// TIA Portal V15.1 export
// export: Created 2020-12-23T12:53:55.1483535Z, ExportSetting WithDefaults, WithReadOnly, DisplayName Totally Integrated Automation Portal, DisplayVersion V15.1 Update 3, DisplayName TIA Portal Openness, DisplayVersion V15.1, DisplayName STEP 7 Professional, DisplayVersion V15.1 Update 3, DisplayName WinCC Advanced, DisplayVersion V15.1 Update 3
FUNCTION "func_outputs" : Void   // FC1331, LAD
TITLE = OUTPUTS
{ S7_Optimized_Access := 'TRUE' }
VERSION : 0.1
// stored: AutoNumber false, CodeModifiedDate 2020-12-23T12:53:21.0067533Z, CompileDate 2020-12-23T12:53:51.673862Z, CreationDate 2020-12-23T07:31:02.6354064Z, HandleErrorsWithinBlock false, InterfaceModifiedDate 2020-12-23T12:48:47.2749857Z, IsConsistent true, IsIECCheckEnabled false, IsKnowHowProtected false, IsWriteProtected false, LibraryConformanceStatus The object is library-conformant., ModifiedDate 2020-12-23T12:53:38.1882563Z, ParameterModified 2020-12-23T07:31:02.6354064Z, PLCSimAdvancedSupport false, SetENOAutomatically False, StructureModified 2020-12-23T07:31:02.6354064Z, UDAEnableTagReadback false
BEGIN

REGION Network 1: ------ [1] TBL TABLE LH ------
   // TABLE LH
END_REGION

REGION Network 2: TBL TABLE LH HP UP
   // CONDICIONES DE SEGURIDAD / WARUNKI BEZPIECZENSTWA
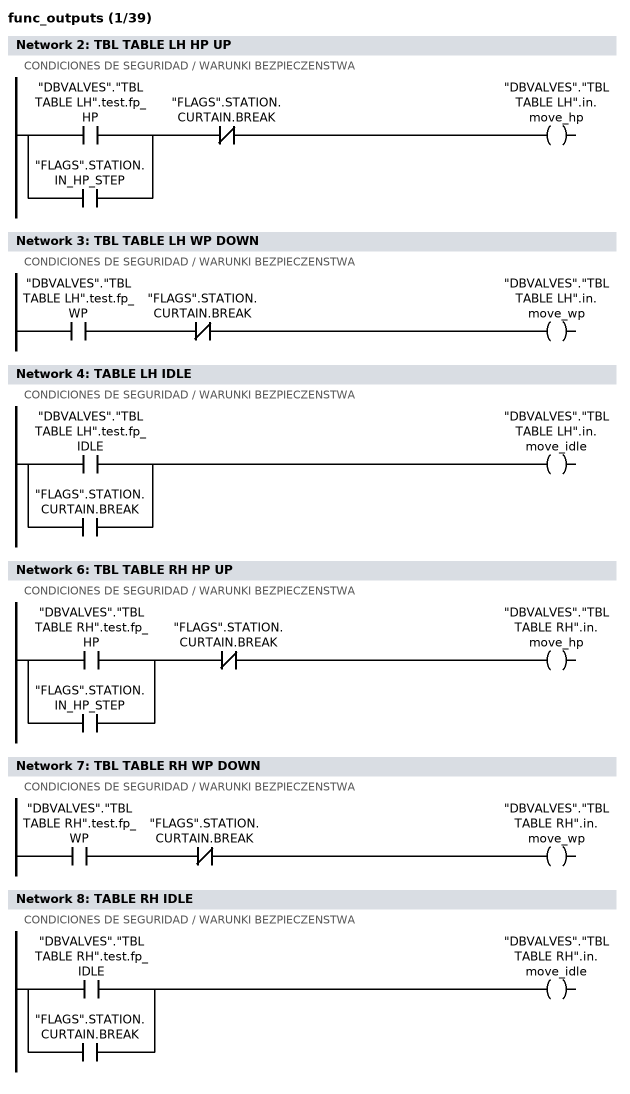
   RUNG wire#powerrail
      Contact( "DBVALVES"."TBL TABLE LH".test.fp_HP )
      wire#w1
      I_Contact( "FLAGS".STATION.CURTAIN.BREAK )
      Coil( "DBVALVES"."TBL TABLE LH".in.move_hp )
   END_RUNG
   RUNG wire#powerrail
      Contact( "FLAGS".STATION.IN_HP_STEP )
   END_RUNG wire#w1
   // the same network as SCL:
   "DBVALVES"."TBL TABLE LH".in.move_hp := ("DBVALVES"."TBL TABLE LH".test.fp_HP OR "FLAGS".STATION.IN_HP_STEP) AND NOT "FLAGS".STATION.CURTAIN.BREAK;
END_REGION

REGION Network 3: TBL TABLE LH WP DOWN
   // CONDICIONES DE SEGURIDAD / WARUNKI BEZPIECZENSTWA
   RUNG wire#powerrail
      Contact( "DBVALVES"."TBL TABLE LH".test.fp_WP )
      I_Contact( "FLAGS".STATION.CURTAIN.BREAK )
      Coil( "DBVALVES"."TBL TABLE LH".in.move_wp )
   END_RUNG
   // the same network as SCL:
   "DBVALVES"."TBL TABLE LH".in.move_wp := "DBVALVES"."TBL TABLE LH".test.fp_WP AND NOT "FLAGS".STATION.CURTAIN.BREAK;
END_REGION

REGION Network 4: TABLE LH IDLE
   // CONDICIONES DE SEGURIDAD / WARUNKI BEZPIECZENSTWA
   RUNG wire#powerrail
      Contact( "DBVALVES"."TBL TABLE LH".test.fp_IDLE )
      wire#w1
      Coil( "DBVALVES"."TBL TABLE LH".in.move_idle )
   END_RUNG
   RUNG wire#powerrail
      Contact( "FLAGS".STATION.CURTAIN.BREAK )
   END_RUNG wire#w1
   // the same network as SCL:
   "DBVALVES"."TBL TABLE LH".in.move_idle := "DBVALVES"."TBL TABLE LH".test.fp_IDLE OR "FLAGS".STATION.CURTAIN.BREAK;
END_REGION

REGION Network 5: ------ [2] TBL TABLE RH ------
   // TABLE RH
END_REGION

REGION Network 6: TBL TABLE RH HP UP
   // CONDICIONES DE SEGURIDAD / WARUNKI BEZPIECZENSTWA
   RUNG wire#powerrail
      Contact( "DBVALVES"."TBL TABLE RH".test.fp_HP )
      wire#w1
      I_Contact( "FLAGS".STATION.CURTAIN.BREAK )
      Coil( "DBVALVES"."TBL TABLE RH".in.move_hp )
   END_RUNG
   RUNG wire#powerrail
      Contact( "FLAGS".STATION.IN_HP_STEP )
   END_RUNG wire#w1
   // the same network as SCL:
   "DBVALVES"."TBL TABLE RH".in.move_hp := ("DBVALVES"."TBL TABLE RH".test.fp_HP OR "FLAGS".STATION.IN_HP_STEP) AND NOT "FLAGS".STATION.CURTAIN.BREAK;
END_REGION

REGION Network 7: TBL TABLE RH WP DOWN
   // CONDICIONES DE SEGURIDAD / WARUNKI BEZPIECZENSTWA
   RUNG wire#powerrail
      Contact( "DBVALVES"."TBL TABLE RH".test.fp_WP )
      I_Contact( "FLAGS".STATION.CURTAIN.BREAK )
      Coil( "DBVALVES"."TBL TABLE RH".in.move_wp )
   END_RUNG
   // the same network as SCL:
   "DBVALVES"."TBL TABLE RH".in.move_wp := "DBVALVES"."TBL TABLE RH".test.fp_WP AND NOT "FLAGS".STATION.CURTAIN.BREAK;
END_REGION

REGION Network 8: TABLE RH IDLE
   // CONDICIONES DE SEGURIDAD / WARUNKI BEZPIECZENSTWA
   RUNG wire#powerrail
      Contact( "DBVALVES"."TBL TABLE RH".test.fp_IDLE )
      wire#w1
      Coil( "DBVALVES"."TBL TABLE RH".in.move_idle )
   END_RUNG
   RUNG wire#powerrail
      Contact( "FLAGS".STATION.CURTAIN.BREAK )
   END_RUNG wire#w1
   // the same network as SCL:
   "DBVALVES"."TBL TABLE RH".in.move_idle := "DBVALVES"."TBL TABLE RH".test.fp_IDLE OR "FLAGS".STATION.CURTAIN.BREAK;
END_REGION

REGION Network 9: ------ [3] TBL SECTION1 ------
   // SECTION1
END_REGION

REGION Network 10: TBL SECTION1 HP UP
   // CONDICIONES DE SEGURIDAD / WARUNKI BEZPIECZENSTWA
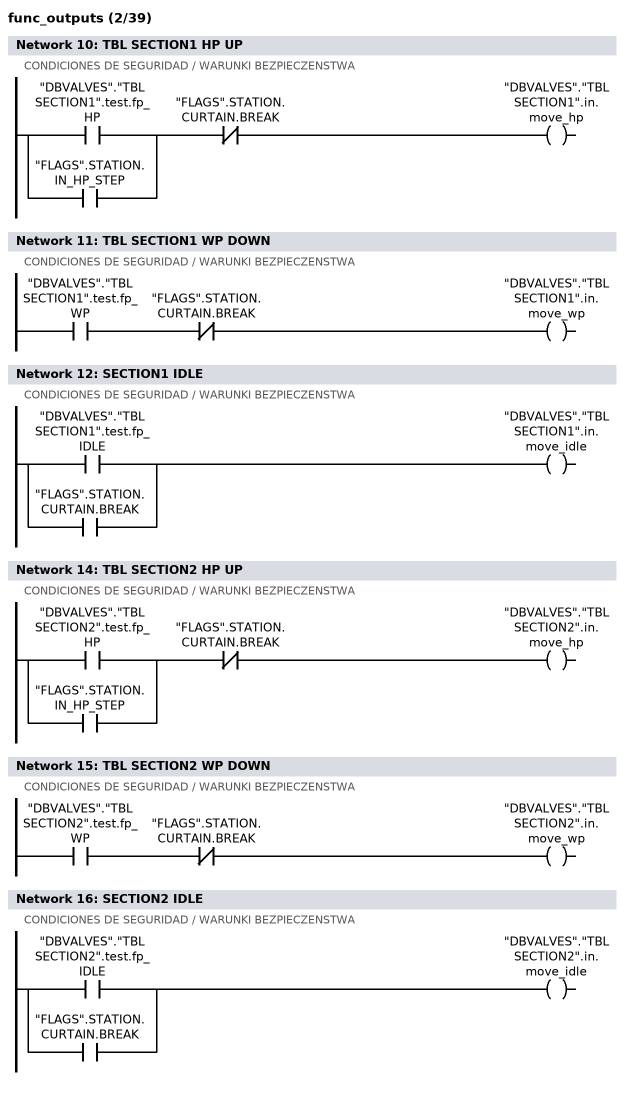
   RUNG wire#powerrail
      Contact( "DBVALVES"."TBL SECTION1".test.fp_HP )
      wire#w1
      I_Contact( "FLAGS".STATION.CURTAIN.BREAK )
      Coil( "DBVALVES"."TBL SECTION1".in.move_hp )
   END_RUNG
   RUNG wire#powerrail
      Contact( "FLAGS".STATION.IN_HP_STEP )
   END_RUNG wire#w1
   // the same network as SCL:
   "DBVALVES"."TBL SECTION1".in.move_hp := ("DBVALVES"."TBL SECTION1".test.fp_HP OR "FLAGS".STATION.IN_HP_STEP) AND NOT "FLAGS".STATION.CURTAIN.BREAK;
END_REGION

REGION Network 11: TBL SECTION1 WP DOWN
   // CONDICIONES DE SEGURIDAD / WARUNKI BEZPIECZENSTWA
   RUNG wire#powerrail
      Contact( "DBVALVES"."TBL SECTION1".test.fp_WP )
      I_Contact( "FLAGS".STATION.CURTAIN.BREAK )
      Coil( "DBVALVES"."TBL SECTION1".in.move_wp )
   END_RUNG
   // the same network as SCL:
   "DBVALVES"."TBL SECTION1".in.move_wp := "DBVALVES"."TBL SECTION1".test.fp_WP AND NOT "FLAGS".STATION.CURTAIN.BREAK;
END_REGION

REGION Network 12: SECTION1 IDLE
   // CONDICIONES DE SEGURIDAD / WARUNKI BEZPIECZENSTWA
   RUNG wire#powerrail
      Contact( "DBVALVES"."TBL SECTION1".test.fp_IDLE )
      wire#w1
      Coil( "DBVALVES"."TBL SECTION1".in.move_idle )
   END_RUNG
   RUNG wire#powerrail
      Contact( "FLAGS".STATION.CURTAIN.BREAK )
   END_RUNG wire#w1
   // the same network as SCL:
   "DBVALVES"."TBL SECTION1".in.move_idle := "DBVALVES"."TBL SECTION1".test.fp_IDLE OR "FLAGS".STATION.CURTAIN.BREAK;
END_REGION

REGION Network 13: ------ [4] TBL SECTION2 ------
   // SECTION2
END_REGION

REGION Network 14: TBL SECTION2 HP UP
   // CONDICIONES DE SEGURIDAD / WARUNKI BEZPIECZENSTWA
   RUNG wire#powerrail
      Contact( "DBVALVES"."TBL SECTION2".test.fp_HP )
      wire#w1
      I_Contact( "FLAGS".STATION.CURTAIN.BREAK )
      Coil( "DBVALVES"."TBL SECTION2".in.move_hp )
   END_RUNG
   RUNG wire#powerrail
      Contact( "FLAGS".STATION.IN_HP_STEP )
   END_RUNG wire#w1
   // the same network as SCL:
   "DBVALVES"."TBL SECTION2".in.move_hp := ("DBVALVES"."TBL SECTION2".test.fp_HP OR "FLAGS".STATION.IN_HP_STEP) AND NOT "FLAGS".STATION.CURTAIN.BREAK;
END_REGION

REGION Network 15: TBL SECTION2 WP DOWN
   // CONDICIONES DE SEGURIDAD / WARUNKI BEZPIECZENSTWA
   RUNG wire#powerrail
      Contact( "DBVALVES"."TBL SECTION2".test.fp_WP )
      I_Contact( "FLAGS".STATION.CURTAIN.BREAK )
      Coil( "DBVALVES"."TBL SECTION2".in.move_wp )
   END_RUNG
   // the same network as SCL:
   "DBVALVES"."TBL SECTION2".in.move_wp := "DBVALVES"."TBL SECTION2".test.fp_WP AND NOT "FLAGS".STATION.CURTAIN.BREAK;
END_REGION

REGION Network 16: SECTION2 IDLE
   // CONDICIONES DE SEGURIDAD / WARUNKI BEZPIECZENSTWA
   RUNG wire#powerrail
      Contact( "DBVALVES"."TBL SECTION2".test.fp_IDLE )
      wire#w1
      Coil( "DBVALVES"."TBL SECTION2".in.move_idle )
   END_RUNG
   RUNG wire#powerrail
      Contact( "FLAGS".STATION.CURTAIN.BREAK )
   END_RUNG wire#w1
   // the same network as SCL:
   "DBVALVES"."TBL SECTION2".in.move_idle := "DBVALVES"."TBL SECTION2".test.fp_IDLE OR "FLAGS".STATION.CURTAIN.BREAK;
END_REGION

REGION Network 17: ------ [5] TBL SECTION4 LH ------
   // SECTION4 LH
END_REGION

REGION Network 18: TBL SECTION4 LH HP UP
   // CONDICIONES DE SEGURIDAD / WARUNKI BEZPIECZENSTWA
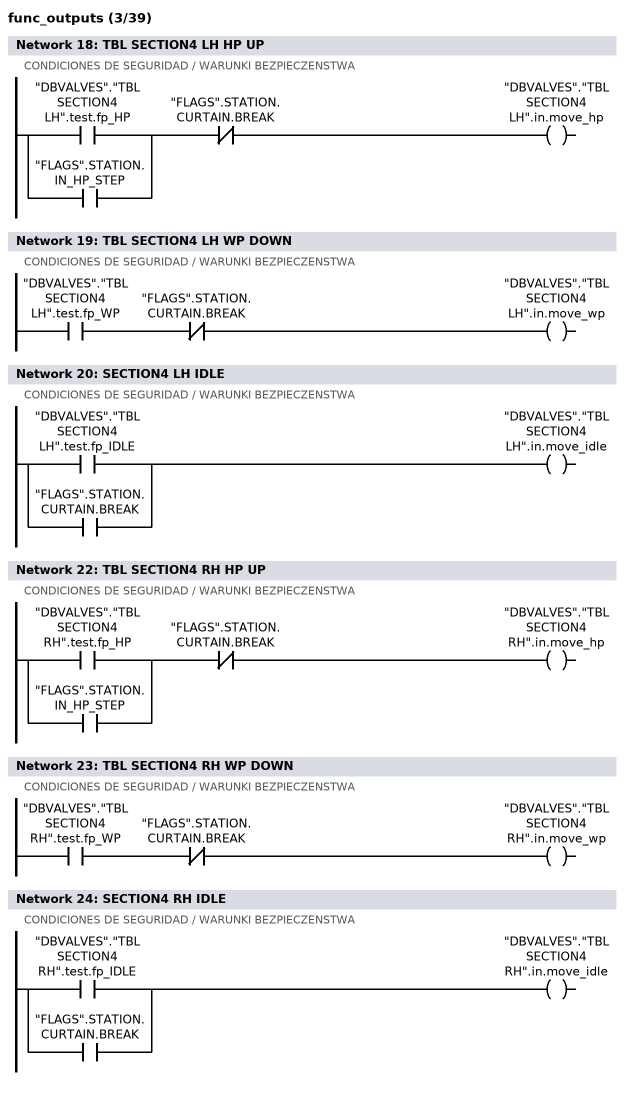
   RUNG wire#powerrail
      Contact( "DBVALVES"."TBL SECTION4 LH".test.fp_HP )
      wire#w1
      I_Contact( "FLAGS".STATION.CURTAIN.BREAK )
      Coil( "DBVALVES"."TBL SECTION4 LH".in.move_hp )
   END_RUNG
   RUNG wire#powerrail
      Contact( "FLAGS".STATION.IN_HP_STEP )
   END_RUNG wire#w1
   // the same network as SCL:
   "DBVALVES"."TBL SECTION4 LH".in.move_hp := ("DBVALVES"."TBL SECTION4 LH".test.fp_HP OR "FLAGS".STATION.IN_HP_STEP) AND NOT "FLAGS".STATION.CURTAIN.BREAK;
END_REGION

REGION Network 19: TBL SECTION4 LH WP DOWN
   // CONDICIONES DE SEGURIDAD / WARUNKI BEZPIECZENSTWA
   RUNG wire#powerrail
      Contact( "DBVALVES"."TBL SECTION4 LH".test.fp_WP )
      I_Contact( "FLAGS".STATION.CURTAIN.BREAK )
      Coil( "DBVALVES"."TBL SECTION4 LH".in.move_wp )
   END_RUNG
   // the same network as SCL:
   "DBVALVES"."TBL SECTION4 LH".in.move_wp := "DBVALVES"."TBL SECTION4 LH".test.fp_WP AND NOT "FLAGS".STATION.CURTAIN.BREAK;
END_REGION

REGION Network 20: SECTION4 LH IDLE
   // CONDICIONES DE SEGURIDAD / WARUNKI BEZPIECZENSTWA
   RUNG wire#powerrail
      Contact( "DBVALVES"."TBL SECTION4 LH".test.fp_IDLE )
      wire#w1
      Coil( "DBVALVES"."TBL SECTION4 LH".in.move_idle )
   END_RUNG
   RUNG wire#powerrail
      Contact( "FLAGS".STATION.CURTAIN.BREAK )
   END_RUNG wire#w1
   // the same network as SCL:
   "DBVALVES"."TBL SECTION4 LH".in.move_idle := "DBVALVES"."TBL SECTION4 LH".test.fp_IDLE OR "FLAGS".STATION.CURTAIN.BREAK;
END_REGION

REGION Network 21: ------ [6] TBL SECTION4 RH ------
   // SECTION4 RH
END_REGION

REGION Network 22: TBL SECTION4 RH HP UP
   // CONDICIONES DE SEGURIDAD / WARUNKI BEZPIECZENSTWA
   RUNG wire#powerrail
      Contact( "DBVALVES"."TBL SECTION4 RH".test.fp_HP )
      wire#w1
      I_Contact( "FLAGS".STATION.CURTAIN.BREAK )
      Coil( "DBVALVES"."TBL SECTION4 RH".in.move_hp )
   END_RUNG
   RUNG wire#powerrail
      Contact( "FLAGS".STATION.IN_HP_STEP )
   END_RUNG wire#w1
   // the same network as SCL:
   "DBVALVES"."TBL SECTION4 RH".in.move_hp := ("DBVALVES"."TBL SECTION4 RH".test.fp_HP OR "FLAGS".STATION.IN_HP_STEP) AND NOT "FLAGS".STATION.CURTAIN.BREAK;
END_REGION

REGION Network 23: TBL SECTION4 RH WP DOWN
   // CONDICIONES DE SEGURIDAD / WARUNKI BEZPIECZENSTWA
   RUNG wire#powerrail
      Contact( "DBVALVES"."TBL SECTION4 RH".test.fp_WP )
      I_Contact( "FLAGS".STATION.CURTAIN.BREAK )
      Coil( "DBVALVES"."TBL SECTION4 RH".in.move_wp )
   END_RUNG
   // the same network as SCL:
   "DBVALVES"."TBL SECTION4 RH".in.move_wp := "DBVALVES"."TBL SECTION4 RH".test.fp_WP AND NOT "FLAGS".STATION.CURTAIN.BREAK;
END_REGION

REGION Network 24: SECTION4 RH IDLE
   // CONDICIONES DE SEGURIDAD / WARUNKI BEZPIECZENSTWA
   RUNG wire#powerrail
      Contact( "DBVALVES"."TBL SECTION4 RH".test.fp_IDLE )
      wire#w1
      Coil( "DBVALVES"."TBL SECTION4 RH".in.move_idle )
   END_RUNG
   RUNG wire#powerrail
      Contact( "FLAGS".STATION.CURTAIN.BREAK )
   END_RUNG wire#w1
   // the same network as SCL:
   "DBVALVES"."TBL SECTION4 RH".in.move_idle := "DBVALVES"."TBL SECTION4 RH".test.fp_IDLE OR "FLAGS".STATION.CURTAIN.BREAK;
END_REGION

REGION Network 25: ------ [7] TBL SECTION5 LH ------
   // SECTION5 LH
END_REGION

REGION Network 26: TBL SECTION5 LH HP UP
   // CONDICIONES DE SEGURIDAD / WARUNKI BEZPIECZENSTWA
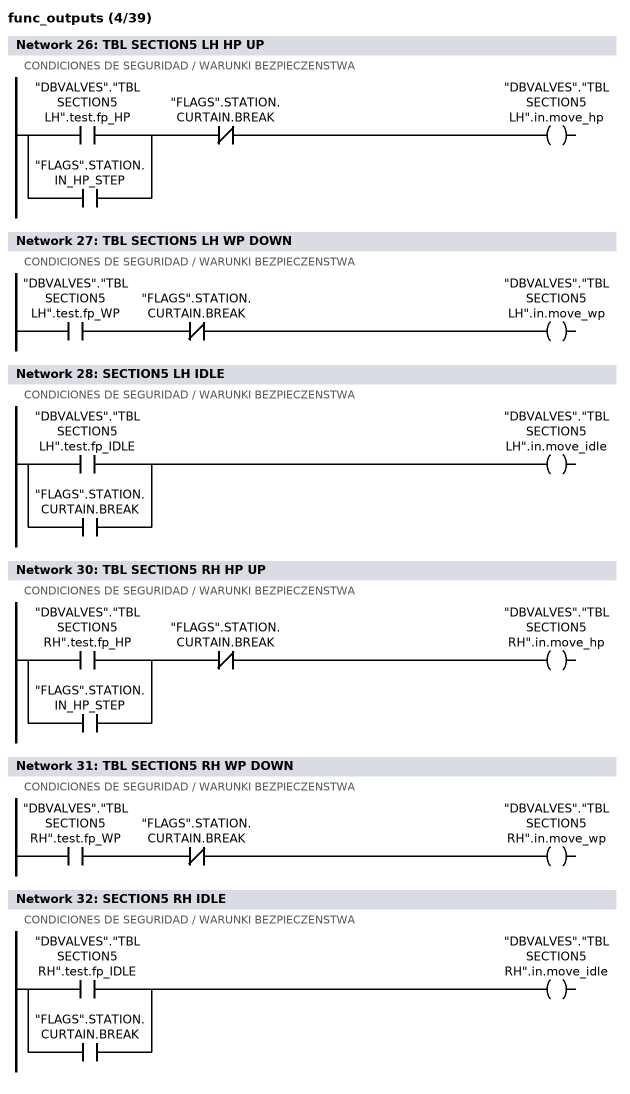
   RUNG wire#powerrail
      Contact( "DBVALVES"."TBL SECTION5 LH".test.fp_HP )
      wire#w1
      I_Contact( "FLAGS".STATION.CURTAIN.BREAK )
      Coil( "DBVALVES"."TBL SECTION5 LH".in.move_hp )
   END_RUNG
   RUNG wire#powerrail
      Contact( "FLAGS".STATION.IN_HP_STEP )
   END_RUNG wire#w1
   // the same network as SCL:
   "DBVALVES"."TBL SECTION5 LH".in.move_hp := ("DBVALVES"."TBL SECTION5 LH".test.fp_HP OR "FLAGS".STATION.IN_HP_STEP) AND NOT "FLAGS".STATION.CURTAIN.BREAK;
END_REGION

REGION Network 27: TBL SECTION5 LH WP DOWN
   // CONDICIONES DE SEGURIDAD / WARUNKI BEZPIECZENSTWA
   RUNG wire#powerrail
      Contact( "DBVALVES"."TBL SECTION5 LH".test.fp_WP )
      I_Contact( "FLAGS".STATION.CURTAIN.BREAK )
      Coil( "DBVALVES"."TBL SECTION5 LH".in.move_wp )
   END_RUNG
   // the same network as SCL:
   "DBVALVES"."TBL SECTION5 LH".in.move_wp := "DBVALVES"."TBL SECTION5 LH".test.fp_WP AND NOT "FLAGS".STATION.CURTAIN.BREAK;
END_REGION

REGION Network 28: SECTION5 LH IDLE
   // CONDICIONES DE SEGURIDAD / WARUNKI BEZPIECZENSTWA
   RUNG wire#powerrail
      Contact( "DBVALVES"."TBL SECTION5 LH".test.fp_IDLE )
      wire#w1
      Coil( "DBVALVES"."TBL SECTION5 LH".in.move_idle )
   END_RUNG
   RUNG wire#powerrail
      Contact( "FLAGS".STATION.CURTAIN.BREAK )
   END_RUNG wire#w1
   // the same network as SCL:
   "DBVALVES"."TBL SECTION5 LH".in.move_idle := "DBVALVES"."TBL SECTION5 LH".test.fp_IDLE OR "FLAGS".STATION.CURTAIN.BREAK;
END_REGION

REGION Network 29: ------ [8] TBL SECTION5 RH ------
   // SECTION5 RH
END_REGION

REGION Network 30: TBL SECTION5 RH HP UP
   // CONDICIONES DE SEGURIDAD / WARUNKI BEZPIECZENSTWA
   RUNG wire#powerrail
      Contact( "DBVALVES"."TBL SECTION5 RH".test.fp_HP )
      wire#w1
      I_Contact( "FLAGS".STATION.CURTAIN.BREAK )
      Coil( "DBVALVES"."TBL SECTION5 RH".in.move_hp )
   END_RUNG
   RUNG wire#powerrail
      Contact( "FLAGS".STATION.IN_HP_STEP )
   END_RUNG wire#w1
   // the same network as SCL:
   "DBVALVES"."TBL SECTION5 RH".in.move_hp := ("DBVALVES"."TBL SECTION5 RH".test.fp_HP OR "FLAGS".STATION.IN_HP_STEP) AND NOT "FLAGS".STATION.CURTAIN.BREAK;
END_REGION

REGION Network 31: TBL SECTION5 RH WP DOWN
   // CONDICIONES DE SEGURIDAD / WARUNKI BEZPIECZENSTWA
   RUNG wire#powerrail
      Contact( "DBVALVES"."TBL SECTION5 RH".test.fp_WP )
      I_Contact( "FLAGS".STATION.CURTAIN.BREAK )
      Coil( "DBVALVES"."TBL SECTION5 RH".in.move_wp )
   END_RUNG
   // the same network as SCL:
   "DBVALVES"."TBL SECTION5 RH".in.move_wp := "DBVALVES"."TBL SECTION5 RH".test.fp_WP AND NOT "FLAGS".STATION.CURTAIN.BREAK;
END_REGION

REGION Network 32: SECTION5 RH IDLE
   // CONDICIONES DE SEGURIDAD / WARUNKI BEZPIECZENSTWA
   RUNG wire#powerrail
      Contact( "DBVALVES"."TBL SECTION5 RH".test.fp_IDLE )
      wire#w1
      Coil( "DBVALVES"."TBL SECTION5 RH".in.move_idle )
   END_RUNG
   RUNG wire#powerrail
      Contact( "FLAGS".STATION.CURTAIN.BREAK )
   END_RUNG wire#w1
   // the same network as SCL:
   "DBVALVES"."TBL SECTION5 RH".in.move_idle := "DBVALVES"."TBL SECTION5 RH".test.fp_IDLE OR "FLAGS".STATION.CURTAIN.BREAK;
END_REGION

REGION Network 33: ------ [9] TBL POSITIONING LH ------
   // POSITIONING LH
END_REGION

REGION Network 34: TBL POSITIONING LH HP UP
   // CONDICIONES DE SEGURIDAD / WARUNKI BEZPIECZENSTWA
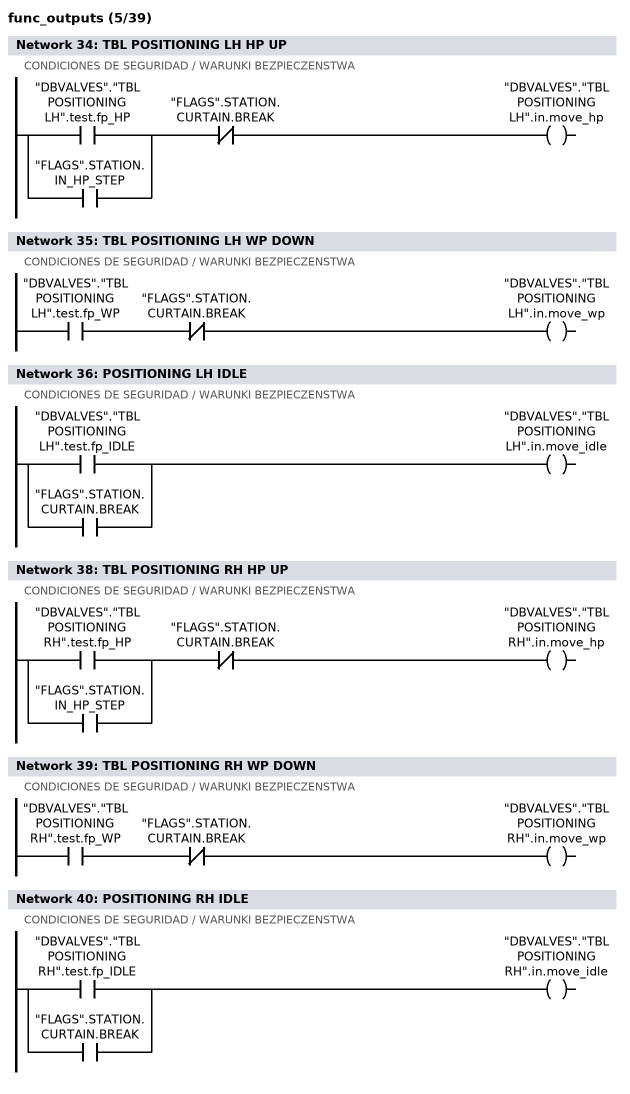
   RUNG wire#powerrail
      Contact( "DBVALVES"."TBL POSITIONING LH".test.fp_HP )
      wire#w1
      I_Contact( "FLAGS".STATION.CURTAIN.BREAK )
      Coil( "DBVALVES"."TBL POSITIONING LH".in.move_hp )
   END_RUNG
   RUNG wire#powerrail
      Contact( "FLAGS".STATION.IN_HP_STEP )
   END_RUNG wire#w1
   // the same network as SCL:
   "DBVALVES"."TBL POSITIONING LH".in.move_hp := ("DBVALVES"."TBL POSITIONING LH".test.fp_HP OR "FLAGS".STATION.IN_HP_STEP) AND NOT "FLAGS".STATION.CURTAIN.BREAK;
END_REGION

REGION Network 35: TBL POSITIONING LH WP DOWN
   // CONDICIONES DE SEGURIDAD / WARUNKI BEZPIECZENSTWA
   RUNG wire#powerrail
      Contact( "DBVALVES"."TBL POSITIONING LH".test.fp_WP )
      I_Contact( "FLAGS".STATION.CURTAIN.BREAK )
      Coil( "DBVALVES"."TBL POSITIONING LH".in.move_wp )
   END_RUNG
   // the same network as SCL:
   "DBVALVES"."TBL POSITIONING LH".in.move_wp := "DBVALVES"."TBL POSITIONING LH".test.fp_WP AND NOT "FLAGS".STATION.CURTAIN.BREAK;
END_REGION

REGION Network 36: POSITIONING LH IDLE
   // CONDICIONES DE SEGURIDAD / WARUNKI BEZPIECZENSTWA
   RUNG wire#powerrail
      Contact( "DBVALVES"."TBL POSITIONING LH".test.fp_IDLE )
      wire#w1
      Coil( "DBVALVES"."TBL POSITIONING LH".in.move_idle )
   END_RUNG
   RUNG wire#powerrail
      Contact( "FLAGS".STATION.CURTAIN.BREAK )
   END_RUNG wire#w1
   // the same network as SCL:
   "DBVALVES"."TBL POSITIONING LH".in.move_idle := "DBVALVES"."TBL POSITIONING LH".test.fp_IDLE OR "FLAGS".STATION.CURTAIN.BREAK;
END_REGION

REGION Network 37: ------ [10] TBL POSITIONING RH ------
   // POSITIONING RH
END_REGION

REGION Network 38: TBL POSITIONING RH HP UP
   // CONDICIONES DE SEGURIDAD / WARUNKI BEZPIECZENSTWA
   RUNG wire#powerrail
      Contact( "DBVALVES"."TBL POSITIONING RH".test.fp_HP )
      wire#w1
      I_Contact( "FLAGS".STATION.CURTAIN.BREAK )
      Coil( "DBVALVES"."TBL POSITIONING RH".in.move_hp )
   END_RUNG
   RUNG wire#powerrail
      Contact( "FLAGS".STATION.IN_HP_STEP )
   END_RUNG wire#w1
   // the same network as SCL:
   "DBVALVES"."TBL POSITIONING RH".in.move_hp := ("DBVALVES"."TBL POSITIONING RH".test.fp_HP OR "FLAGS".STATION.IN_HP_STEP) AND NOT "FLAGS".STATION.CURTAIN.BREAK;
END_REGION

REGION Network 39: TBL POSITIONING RH WP DOWN
   // CONDICIONES DE SEGURIDAD / WARUNKI BEZPIECZENSTWA
   RUNG wire#powerrail
      Contact( "DBVALVES"."TBL POSITIONING RH".test.fp_WP )
      I_Contact( "FLAGS".STATION.CURTAIN.BREAK )
      Coil( "DBVALVES"."TBL POSITIONING RH".in.move_wp )
   END_RUNG
   // the same network as SCL:
   "DBVALVES"."TBL POSITIONING RH".in.move_wp := "DBVALVES"."TBL POSITIONING RH".test.fp_WP AND NOT "FLAGS".STATION.CURTAIN.BREAK;
END_REGION

REGION Network 40: POSITIONING RH IDLE
   // CONDICIONES DE SEGURIDAD / WARUNKI BEZPIECZENSTWA
   RUNG wire#powerrail
      Contact( "DBVALVES"."TBL POSITIONING RH".test.fp_IDLE )
      wire#w1
      Coil( "DBVALVES"."TBL POSITIONING RH".in.move_idle )
   END_RUNG
   RUNG wire#powerrail
      Contact( "FLAGS".STATION.CURTAIN.BREAK )
   END_RUNG wire#w1
   // the same network as SCL:
   "DBVALVES"."TBL POSITIONING RH".in.move_idle := "DBVALVES"."TBL POSITIONING RH".test.fp_IDLE OR "FLAGS".STATION.CURTAIN.BREAK;
END_REGION

REGION Network 41: ------ [11] TBL PIN LH ------
   // PIN LH
END_REGION

REGION Network 42: TBL PIN LH HP DOWN
   // CONDICIONES DE SEGURIDAD / WARUNKI BEZPIECZENSTWA
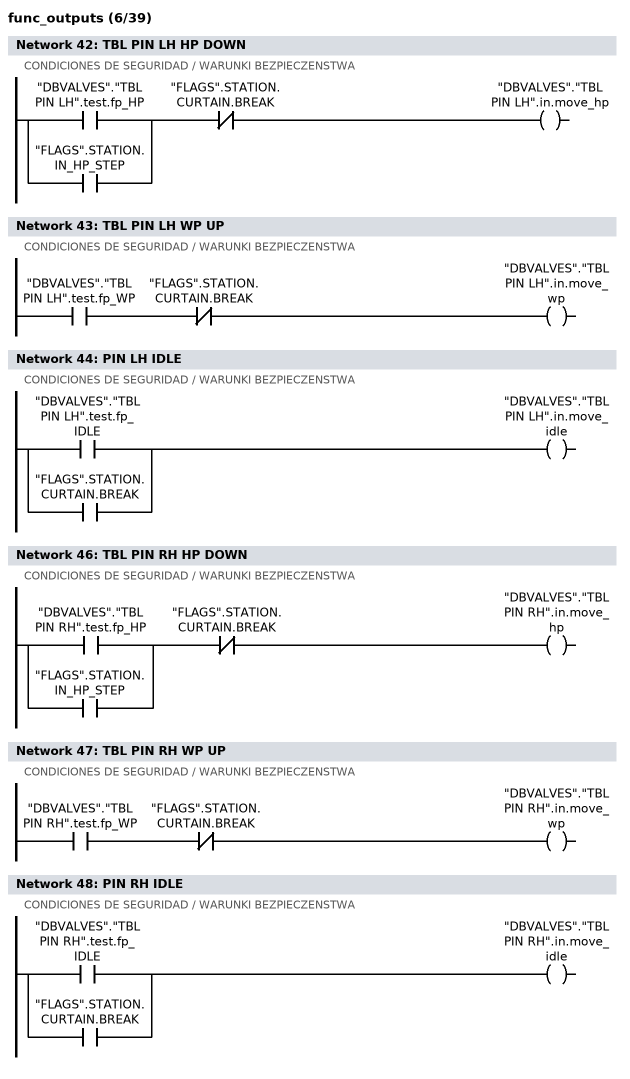
   RUNG wire#powerrail
      Contact( "DBVALVES"."TBL PIN LH".test.fp_HP )
      wire#w1
      I_Contact( "FLAGS".STATION.CURTAIN.BREAK )
      Coil( "DBVALVES"."TBL PIN LH".in.move_hp )
   END_RUNG
   RUNG wire#powerrail
      Contact( "FLAGS".STATION.IN_HP_STEP )
   END_RUNG wire#w1
   // the same network as SCL:
   "DBVALVES"."TBL PIN LH".in.move_hp := ("DBVALVES"."TBL PIN LH".test.fp_HP OR "FLAGS".STATION.IN_HP_STEP) AND NOT "FLAGS".STATION.CURTAIN.BREAK;
END_REGION

REGION Network 43: TBL PIN LH WP UP
   // CONDICIONES DE SEGURIDAD / WARUNKI BEZPIECZENSTWA
   RUNG wire#powerrail
      Contact( "DBVALVES"."TBL PIN LH".test.fp_WP )
      I_Contact( "FLAGS".STATION.CURTAIN.BREAK )
      Coil( "DBVALVES"."TBL PIN LH".in.move_wp )
   END_RUNG
   // the same network as SCL:
   "DBVALVES"."TBL PIN LH".in.move_wp := "DBVALVES"."TBL PIN LH".test.fp_WP AND NOT "FLAGS".STATION.CURTAIN.BREAK;
END_REGION

REGION Network 44: PIN LH IDLE
   // CONDICIONES DE SEGURIDAD / WARUNKI BEZPIECZENSTWA
   RUNG wire#powerrail
      Contact( "DBVALVES"."TBL PIN LH".test.fp_IDLE )
      wire#w1
      Coil( "DBVALVES"."TBL PIN LH".in.move_idle )
   END_RUNG
   RUNG wire#powerrail
      Contact( "FLAGS".STATION.CURTAIN.BREAK )
   END_RUNG wire#w1
   // the same network as SCL:
   "DBVALVES"."TBL PIN LH".in.move_idle := "DBVALVES"."TBL PIN LH".test.fp_IDLE OR "FLAGS".STATION.CURTAIN.BREAK;
END_REGION

REGION Network 45: ------ [12] TBL PIN RH ------
   // PIN RH
END_REGION

REGION Network 46: TBL PIN RH HP DOWN
   // CONDICIONES DE SEGURIDAD / WARUNKI BEZPIECZENSTWA
   RUNG wire#powerrail
      Contact( "DBVALVES"."TBL PIN RH".test.fp_HP )
      wire#w1
      I_Contact( "FLAGS".STATION.CURTAIN.BREAK )
      Coil( "DBVALVES"."TBL PIN RH".in.move_hp )
   END_RUNG
   RUNG wire#powerrail
      Contact( "FLAGS".STATION.IN_HP_STEP )
   END_RUNG wire#w1
   // the same network as SCL:
   "DBVALVES"."TBL PIN RH".in.move_hp := ("DBVALVES"."TBL PIN RH".test.fp_HP OR "FLAGS".STATION.IN_HP_STEP) AND NOT "FLAGS".STATION.CURTAIN.BREAK;
END_REGION

REGION Network 47: TBL PIN RH WP UP
   // CONDICIONES DE SEGURIDAD / WARUNKI BEZPIECZENSTWA
   RUNG wire#powerrail
      Contact( "DBVALVES"."TBL PIN RH".test.fp_WP )
      I_Contact( "FLAGS".STATION.CURTAIN.BREAK )
      Coil( "DBVALVES"."TBL PIN RH".in.move_wp )
   END_RUNG
   // the same network as SCL:
   "DBVALVES"."TBL PIN RH".in.move_wp := "DBVALVES"."TBL PIN RH".test.fp_WP AND NOT "FLAGS".STATION.CURTAIN.BREAK;
END_REGION

REGION Network 48: PIN RH IDLE
   // CONDICIONES DE SEGURIDAD / WARUNKI BEZPIECZENSTWA
   RUNG wire#powerrail
      Contact( "DBVALVES"."TBL PIN RH".test.fp_IDLE )
      wire#w1
      Coil( "DBVALVES"."TBL PIN RH".in.move_idle )
   END_RUNG
   RUNG wire#powerrail
      Contact( "FLAGS".STATION.CURTAIN.BREAK )
   END_RUNG wire#w1
   // the same network as SCL:
   "DBVALVES"."TBL PIN RH".in.move_idle := "DBVALVES"."TBL PIN RH".test.fp_IDLE OR "FLAGS".STATION.CURTAIN.BREAK;
END_REGION

REGION Network 49: ------ [13] TBL SCREW GRIPPER ------
   // SCREW GRIPPER
END_REGION

REGION Network 50: TBL SCREW GRIPPER HP OPEN
   // CONDICIONES DE SEGURIDAD / WARUNKI BEZPIECZENSTWA
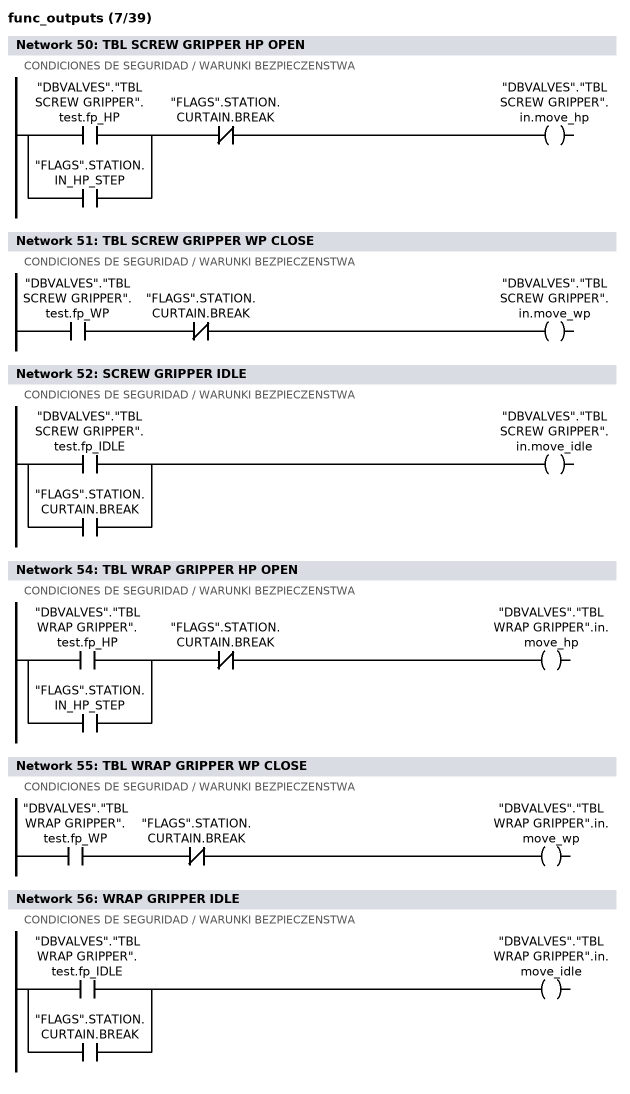
   RUNG wire#powerrail
      Contact( "DBVALVES"."TBL SCREW GRIPPER".test.fp_HP )
      wire#w1
      I_Contact( "FLAGS".STATION.CURTAIN.BREAK )
      Coil( "DBVALVES"."TBL SCREW GRIPPER".in.move_hp )
   END_RUNG
   RUNG wire#powerrail
      Contact( "FLAGS".STATION.IN_HP_STEP )
   END_RUNG wire#w1
   // the same network as SCL:
   "DBVALVES"."TBL SCREW GRIPPER".in.move_hp := ("DBVALVES"."TBL SCREW GRIPPER".test.fp_HP OR "FLAGS".STATION.IN_HP_STEP) AND NOT "FLAGS".STATION.CURTAIN.BREAK;
END_REGION

REGION Network 51: TBL SCREW GRIPPER WP CLOSE
   // CONDICIONES DE SEGURIDAD / WARUNKI BEZPIECZENSTWA
   RUNG wire#powerrail
      Contact( "DBVALVES"."TBL SCREW GRIPPER".test.fp_WP )
      I_Contact( "FLAGS".STATION.CURTAIN.BREAK )
      Coil( "DBVALVES"."TBL SCREW GRIPPER".in.move_wp )
   END_RUNG
   // the same network as SCL:
   "DBVALVES"."TBL SCREW GRIPPER".in.move_wp := "DBVALVES"."TBL SCREW GRIPPER".test.fp_WP AND NOT "FLAGS".STATION.CURTAIN.BREAK;
END_REGION

REGION Network 52: SCREW GRIPPER IDLE
   // CONDICIONES DE SEGURIDAD / WARUNKI BEZPIECZENSTWA
   RUNG wire#powerrail
      Contact( "DBVALVES"."TBL SCREW GRIPPER".test.fp_IDLE )
      wire#w1
      Coil( "DBVALVES"."TBL SCREW GRIPPER".in.move_idle )
   END_RUNG
   RUNG wire#powerrail
      Contact( "FLAGS".STATION.CURTAIN.BREAK )
   END_RUNG wire#w1
   // the same network as SCL:
   "DBVALVES"."TBL SCREW GRIPPER".in.move_idle := "DBVALVES"."TBL SCREW GRIPPER".test.fp_IDLE OR "FLAGS".STATION.CURTAIN.BREAK;
END_REGION

REGION Network 53: ------ [14] TBL WRAP GRIPPER ------
   // WRAP GRIPPER
END_REGION

REGION Network 54: TBL WRAP GRIPPER HP OPEN
   // CONDICIONES DE SEGURIDAD / WARUNKI BEZPIECZENSTWA
   RUNG wire#powerrail
      Contact( "DBVALVES"."TBL WRAP GRIPPER".test.fp_HP )
      wire#w1
      I_Contact( "FLAGS".STATION.CURTAIN.BREAK )
      Coil( "DBVALVES"."TBL WRAP GRIPPER".in.move_hp )
   END_RUNG
   RUNG wire#powerrail
      Contact( "FLAGS".STATION.IN_HP_STEP )
   END_RUNG wire#w1
   // the same network as SCL:
   "DBVALVES"."TBL WRAP GRIPPER".in.move_hp := ("DBVALVES"."TBL WRAP GRIPPER".test.fp_HP OR "FLAGS".STATION.IN_HP_STEP) AND NOT "FLAGS".STATION.CURTAIN.BREAK;
END_REGION

REGION Network 55: TBL WRAP GRIPPER WP CLOSE
   // CONDICIONES DE SEGURIDAD / WARUNKI BEZPIECZENSTWA
   RUNG wire#powerrail
      Contact( "DBVALVES"."TBL WRAP GRIPPER".test.fp_WP )
      I_Contact( "FLAGS".STATION.CURTAIN.BREAK )
      Coil( "DBVALVES"."TBL WRAP GRIPPER".in.move_wp )
   END_RUNG
   // the same network as SCL:
   "DBVALVES"."TBL WRAP GRIPPER".in.move_wp := "DBVALVES"."TBL WRAP GRIPPER".test.fp_WP AND NOT "FLAGS".STATION.CURTAIN.BREAK;
END_REGION

REGION Network 56: WRAP GRIPPER IDLE
   // CONDICIONES DE SEGURIDAD / WARUNKI BEZPIECZENSTWA
   RUNG wire#powerrail
      Contact( "DBVALVES"."TBL WRAP GRIPPER".test.fp_IDLE )
      wire#w1
      Coil( "DBVALVES"."TBL WRAP GRIPPER".in.move_idle )
   END_RUNG
   RUNG wire#powerrail
      Contact( "FLAGS".STATION.CURTAIN.BREAK )
   END_RUNG wire#w1
   // the same network as SCL:
   "DBVALVES"."TBL WRAP GRIPPER".in.move_idle := "DBVALVES"."TBL WRAP GRIPPER".test.fp_IDLE OR "FLAGS".STATION.CURTAIN.BREAK;
END_REGION

REGION Network 57: ------ [15] ST1 POSITIONING ------
   // POSITIONING
END_REGION

REGION Network 58: ST1 POSITIONING HP RIGHT
   // CONDICIONES DE SEGURIDAD / WARUNKI BEZPIECZENSTWA
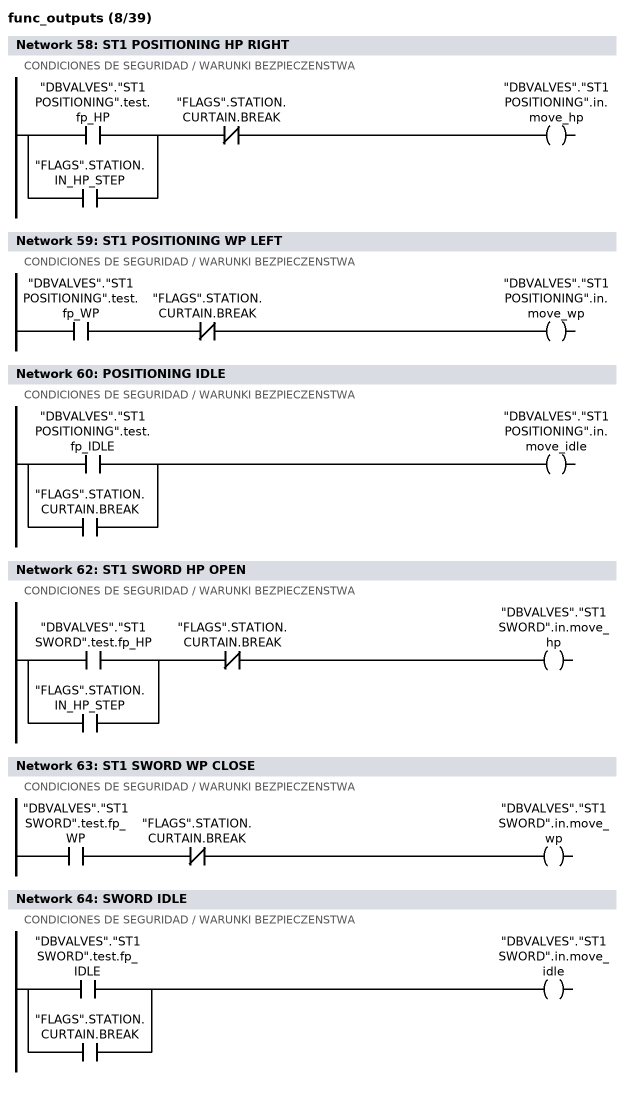
   RUNG wire#powerrail
      Contact( "DBVALVES"."ST1 POSITIONING".test.fp_HP )
      wire#w1
      I_Contact( "FLAGS".STATION.CURTAIN.BREAK )
      Coil( "DBVALVES"."ST1 POSITIONING".in.move_hp )
   END_RUNG
   RUNG wire#powerrail
      Contact( "FLAGS".STATION.IN_HP_STEP )
   END_RUNG wire#w1
   // the same network as SCL:
   "DBVALVES"."ST1 POSITIONING".in.move_hp := ("DBVALVES"."ST1 POSITIONING".test.fp_HP OR "FLAGS".STATION.IN_HP_STEP) AND NOT "FLAGS".STATION.CURTAIN.BREAK;
END_REGION

REGION Network 59: ST1 POSITIONING WP LEFT
   // CONDICIONES DE SEGURIDAD / WARUNKI BEZPIECZENSTWA
   RUNG wire#powerrail
      Contact( "DBVALVES"."ST1 POSITIONING".test.fp_WP )
      I_Contact( "FLAGS".STATION.CURTAIN.BREAK )
      Coil( "DBVALVES"."ST1 POSITIONING".in.move_wp )
   END_RUNG
   // the same network as SCL:
   "DBVALVES"."ST1 POSITIONING".in.move_wp := "DBVALVES"."ST1 POSITIONING".test.fp_WP AND NOT "FLAGS".STATION.CURTAIN.BREAK;
END_REGION

REGION Network 60: POSITIONING IDLE
   // CONDICIONES DE SEGURIDAD / WARUNKI BEZPIECZENSTWA
   RUNG wire#powerrail
      Contact( "DBVALVES"."ST1 POSITIONING".test.fp_IDLE )
      wire#w1
      Coil( "DBVALVES"."ST1 POSITIONING".in.move_idle )
   END_RUNG
   RUNG wire#powerrail
      Contact( "FLAGS".STATION.CURTAIN.BREAK )
   END_RUNG wire#w1
   // the same network as SCL:
   "DBVALVES"."ST1 POSITIONING".in.move_idle := "DBVALVES"."ST1 POSITIONING".test.fp_IDLE OR "FLAGS".STATION.CURTAIN.BREAK;
END_REGION

REGION Network 61: ------ [16] ST1 SWORD ------
   // SWORD
END_REGION

REGION Network 62: ST1 SWORD HP OPEN
   // CONDICIONES DE SEGURIDAD / WARUNKI BEZPIECZENSTWA
   RUNG wire#powerrail
      Contact( "DBVALVES"."ST1 SWORD".test.fp_HP )
      wire#w1
      I_Contact( "FLAGS".STATION.CURTAIN.BREAK )
      Coil( "DBVALVES"."ST1 SWORD".in.move_hp )
   END_RUNG
   RUNG wire#powerrail
      Contact( "FLAGS".STATION.IN_HP_STEP )
   END_RUNG wire#w1
   // the same network as SCL:
   "DBVALVES"."ST1 SWORD".in.move_hp := ("DBVALVES"."ST1 SWORD".test.fp_HP OR "FLAGS".STATION.IN_HP_STEP) AND NOT "FLAGS".STATION.CURTAIN.BREAK;
END_REGION

REGION Network 63: ST1 SWORD WP CLOSE
   // CONDICIONES DE SEGURIDAD / WARUNKI BEZPIECZENSTWA
   RUNG wire#powerrail
      Contact( "DBVALVES"."ST1 SWORD".test.fp_WP )
      I_Contact( "FLAGS".STATION.CURTAIN.BREAK )
      Coil( "DBVALVES"."ST1 SWORD".in.move_wp )
   END_RUNG
   // the same network as SCL:
   "DBVALVES"."ST1 SWORD".in.move_wp := "DBVALVES"."ST1 SWORD".test.fp_WP AND NOT "FLAGS".STATION.CURTAIN.BREAK;
END_REGION

REGION Network 64: SWORD IDLE
   // CONDICIONES DE SEGURIDAD / WARUNKI BEZPIECZENSTWA
   RUNG wire#powerrail
      Contact( "DBVALVES"."ST1 SWORD".test.fp_IDLE )
      wire#w1
      Coil( "DBVALVES"."ST1 SWORD".in.move_idle )
   END_RUNG
   RUNG wire#powerrail
      Contact( "FLAGS".STATION.CURTAIN.BREAK )
   END_RUNG wire#w1
   // the same network as SCL:
   "DBVALVES"."ST1 SWORD".in.move_idle := "DBVALVES"."ST1 SWORD".test.fp_IDLE OR "FLAGS".STATION.CURTAIN.BREAK;
END_REGION

REGION Network 65: ------ [17] ST2 POSITIONING ------
   // POSITIONING
END_REGION

REGION Network 66: ST2 POSITIONING HP BACK
   // CONDICIONES DE SEGURIDAD / WARUNKI BEZPIECZENSTWA
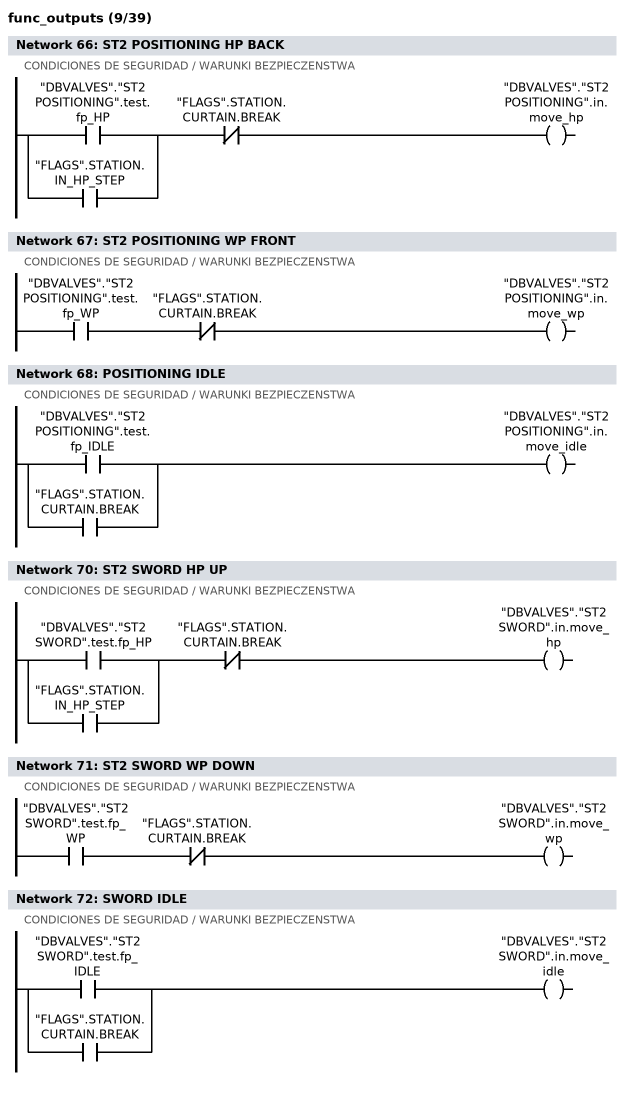
   RUNG wire#powerrail
      Contact( "DBVALVES"."ST2 POSITIONING".test.fp_HP )
      wire#w1
      I_Contact( "FLAGS".STATION.CURTAIN.BREAK )
      Coil( "DBVALVES"."ST2 POSITIONING".in.move_hp )
   END_RUNG
   RUNG wire#powerrail
      Contact( "FLAGS".STATION.IN_HP_STEP )
   END_RUNG wire#w1
   // the same network as SCL:
   "DBVALVES"."ST2 POSITIONING".in.move_hp := ("DBVALVES"."ST2 POSITIONING".test.fp_HP OR "FLAGS".STATION.IN_HP_STEP) AND NOT "FLAGS".STATION.CURTAIN.BREAK;
END_REGION

REGION Network 67: ST2 POSITIONING WP FRONT
   // CONDICIONES DE SEGURIDAD / WARUNKI BEZPIECZENSTWA
   RUNG wire#powerrail
      Contact( "DBVALVES"."ST2 POSITIONING".test.fp_WP )
      I_Contact( "FLAGS".STATION.CURTAIN.BREAK )
      Coil( "DBVALVES"."ST2 POSITIONING".in.move_wp )
   END_RUNG
   // the same network as SCL:
   "DBVALVES"."ST2 POSITIONING".in.move_wp := "DBVALVES"."ST2 POSITIONING".test.fp_WP AND NOT "FLAGS".STATION.CURTAIN.BREAK;
END_REGION

REGION Network 68: POSITIONING IDLE
   // CONDICIONES DE SEGURIDAD / WARUNKI BEZPIECZENSTWA
   RUNG wire#powerrail
      Contact( "DBVALVES"."ST2 POSITIONING".test.fp_IDLE )
      wire#w1
      Coil( "DBVALVES"."ST2 POSITIONING".in.move_idle )
   END_RUNG
   RUNG wire#powerrail
      Contact( "FLAGS".STATION.CURTAIN.BREAK )
   END_RUNG wire#w1
   // the same network as SCL:
   "DBVALVES"."ST2 POSITIONING".in.move_idle := "DBVALVES"."ST2 POSITIONING".test.fp_IDLE OR "FLAGS".STATION.CURTAIN.BREAK;
END_REGION

REGION Network 69: ------ [18] ST2 SWORD ------
   // SWORD
END_REGION

REGION Network 70: ST2 SWORD HP UP
   // CONDICIONES DE SEGURIDAD / WARUNKI BEZPIECZENSTWA
   RUNG wire#powerrail
      Contact( "DBVALVES"."ST2 SWORD".test.fp_HP )
      wire#w1
      I_Contact( "FLAGS".STATION.CURTAIN.BREAK )
      Coil( "DBVALVES"."ST2 SWORD".in.move_hp )
   END_RUNG
   RUNG wire#powerrail
      Contact( "FLAGS".STATION.IN_HP_STEP )
   END_RUNG wire#w1
   // the same network as SCL:
   "DBVALVES"."ST2 SWORD".in.move_hp := ("DBVALVES"."ST2 SWORD".test.fp_HP OR "FLAGS".STATION.IN_HP_STEP) AND NOT "FLAGS".STATION.CURTAIN.BREAK;
END_REGION

REGION Network 71: ST2 SWORD WP DOWN
   // CONDICIONES DE SEGURIDAD / WARUNKI BEZPIECZENSTWA
   RUNG wire#powerrail
      Contact( "DBVALVES"."ST2 SWORD".test.fp_WP )
      I_Contact( "FLAGS".STATION.CURTAIN.BREAK )
      Coil( "DBVALVES"."ST2 SWORD".in.move_wp )
   END_RUNG
   // the same network as SCL:
   "DBVALVES"."ST2 SWORD".in.move_wp := "DBVALVES"."ST2 SWORD".test.fp_WP AND NOT "FLAGS".STATION.CURTAIN.BREAK;
END_REGION

REGION Network 72: SWORD IDLE
   // CONDICIONES DE SEGURIDAD / WARUNKI BEZPIECZENSTWA
   RUNG wire#powerrail
      Contact( "DBVALVES"."ST2 SWORD".test.fp_IDLE )
      wire#w1
      Coil( "DBVALVES"."ST2 SWORD".in.move_idle )
   END_RUNG
   RUNG wire#powerrail
      Contact( "FLAGS".STATION.CURTAIN.BREAK )
   END_RUNG wire#w1
   // the same network as SCL:
   "DBVALVES"."ST2 SWORD".in.move_idle := "DBVALVES"."ST2 SWORD".test.fp_IDLE OR "FLAGS".STATION.CURTAIN.BREAK;
END_REGION

REGION Network 73: ------ [19] ST3 POSITIONING ------
   // POSITIONING
END_REGION

REGION Network 74: ST3 POSITIONING HP BACK
   // CONDICIONES DE SEGURIDAD / WARUNKI BEZPIECZENSTWA
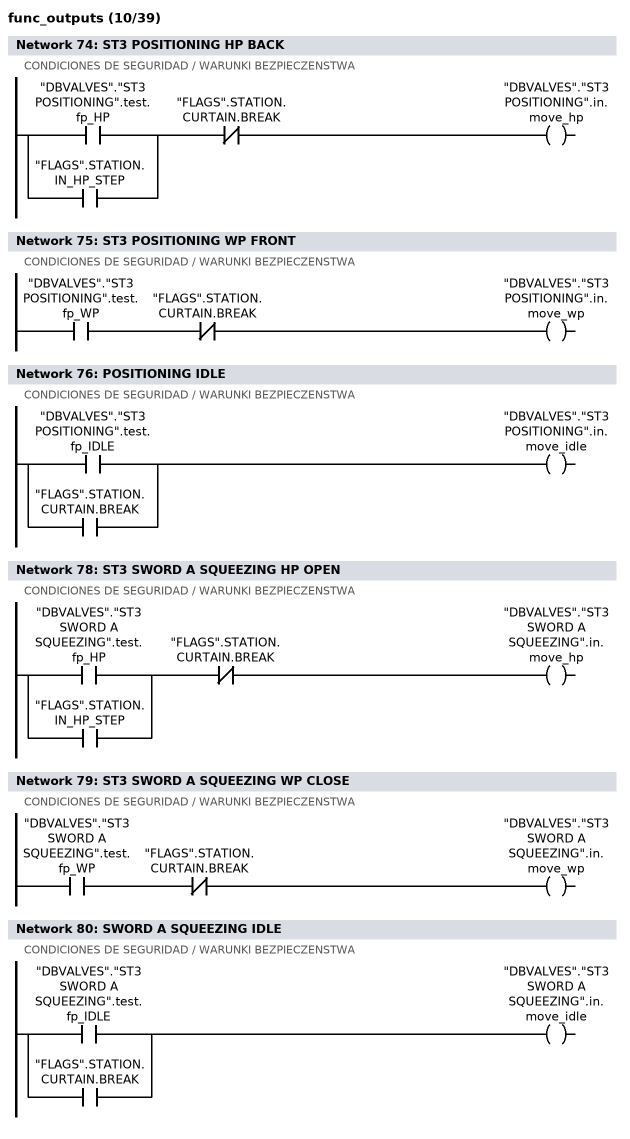
   RUNG wire#powerrail
      Contact( "DBVALVES"."ST3 POSITIONING".test.fp_HP )
      wire#w1
      I_Contact( "FLAGS".STATION.CURTAIN.BREAK )
      Coil( "DBVALVES"."ST3 POSITIONING".in.move_hp )
   END_RUNG
   RUNG wire#powerrail
      Contact( "FLAGS".STATION.IN_HP_STEP )
   END_RUNG wire#w1
   // the same network as SCL:
   "DBVALVES"."ST3 POSITIONING".in.move_hp := ("DBVALVES"."ST3 POSITIONING".test.fp_HP OR "FLAGS".STATION.IN_HP_STEP) AND NOT "FLAGS".STATION.CURTAIN.BREAK;
END_REGION

REGION Network 75: ST3 POSITIONING WP FRONT
   // CONDICIONES DE SEGURIDAD / WARUNKI BEZPIECZENSTWA
   RUNG wire#powerrail
      Contact( "DBVALVES"."ST3 POSITIONING".test.fp_WP )
      I_Contact( "FLAGS".STATION.CURTAIN.BREAK )
      Coil( "DBVALVES"."ST3 POSITIONING".in.move_wp )
   END_RUNG
   // the same network as SCL:
   "DBVALVES"."ST3 POSITIONING".in.move_wp := "DBVALVES"."ST3 POSITIONING".test.fp_WP AND NOT "FLAGS".STATION.CURTAIN.BREAK;
END_REGION

REGION Network 76: POSITIONING IDLE
   // CONDICIONES DE SEGURIDAD / WARUNKI BEZPIECZENSTWA
   RUNG wire#powerrail
      Contact( "DBVALVES"."ST3 POSITIONING".test.fp_IDLE )
      wire#w1
      Coil( "DBVALVES"."ST3 POSITIONING".in.move_idle )
   END_RUNG
   RUNG wire#powerrail
      Contact( "FLAGS".STATION.CURTAIN.BREAK )
   END_RUNG wire#w1
   // the same network as SCL:
   "DBVALVES"."ST3 POSITIONING".in.move_idle := "DBVALVES"."ST3 POSITIONING".test.fp_IDLE OR "FLAGS".STATION.CURTAIN.BREAK;
END_REGION

REGION Network 77: ------ [20] ST3 SWORD A SQUEEZING ------
   // SWORD A SQUEEZING
END_REGION

REGION Network 78: ST3 SWORD A SQUEEZING HP OPEN
   // CONDICIONES DE SEGURIDAD / WARUNKI BEZPIECZENSTWA
   RUNG wire#powerrail
      Contact( "DBVALVES"."ST3 SWORD A SQUEEZING".test.fp_HP )
      wire#w1
      I_Contact( "FLAGS".STATION.CURTAIN.BREAK )
      Coil( "DBVALVES"."ST3 SWORD A SQUEEZING".in.move_hp )
   END_RUNG
   RUNG wire#powerrail
      Contact( "FLAGS".STATION.IN_HP_STEP )
   END_RUNG wire#w1
   // the same network as SCL:
   "DBVALVES"."ST3 SWORD A SQUEEZING".in.move_hp := ("DBVALVES"."ST3 SWORD A SQUEEZING".test.fp_HP OR "FLAGS".STATION.IN_HP_STEP) AND NOT "FLAGS".STATION.CURTAIN.BREAK;
END_REGION

REGION Network 79: ST3 SWORD A SQUEEZING WP CLOSE
   // CONDICIONES DE SEGURIDAD / WARUNKI BEZPIECZENSTWA
   RUNG wire#powerrail
      Contact( "DBVALVES"."ST3 SWORD A SQUEEZING".test.fp_WP )
      I_Contact( "FLAGS".STATION.CURTAIN.BREAK )
      Coil( "DBVALVES"."ST3 SWORD A SQUEEZING".in.move_wp )
   END_RUNG
   // the same network as SCL:
   "DBVALVES"."ST3 SWORD A SQUEEZING".in.move_wp := "DBVALVES"."ST3 SWORD A SQUEEZING".test.fp_WP AND NOT "FLAGS".STATION.CURTAIN.BREAK;
END_REGION

REGION Network 80: SWORD A SQUEEZING IDLE
   // CONDICIONES DE SEGURIDAD / WARUNKI BEZPIECZENSTWA
   RUNG wire#powerrail
      Contact( "DBVALVES"."ST3 SWORD A SQUEEZING".test.fp_IDLE )
      wire#w1
      Coil( "DBVALVES"."ST3 SWORD A SQUEEZING".in.move_idle )
   END_RUNG
   RUNG wire#powerrail
      Contact( "FLAGS".STATION.CURTAIN.BREAK )
   END_RUNG wire#w1
   // the same network as SCL:
   "DBVALVES"."ST3 SWORD A SQUEEZING".in.move_idle := "DBVALVES"."ST3 SWORD A SQUEEZING".test.fp_IDLE OR "FLAGS".STATION.CURTAIN.BREAK;
END_REGION

REGION Network 81: ------ [21] ST3 SWORD A SPREADING ------
   // SWORD A SPREADING
END_REGION

REGION Network 82: ST3 SWORD A SPREADING HP OPEN
   // CONDICIONES DE SEGURIDAD / WARUNKI BEZPIECZENSTWA
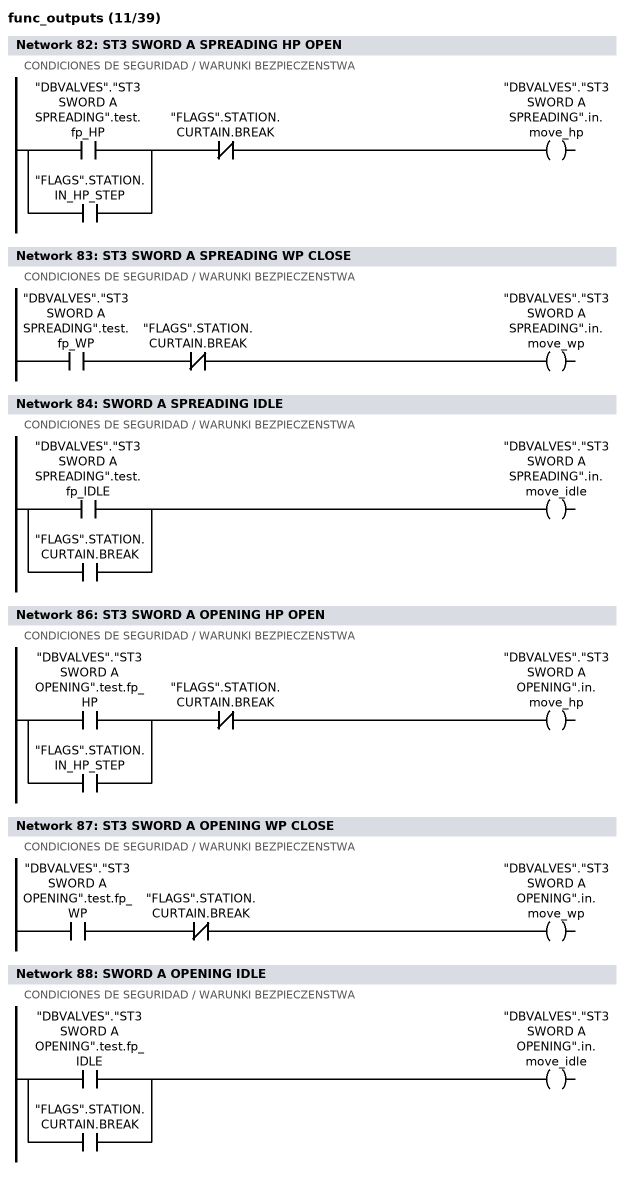
   RUNG wire#powerrail
      Contact( "DBVALVES"."ST3 SWORD A SPREADING".test.fp_HP )
      wire#w1
      I_Contact( "FLAGS".STATION.CURTAIN.BREAK )
      Coil( "DBVALVES"."ST3 SWORD A SPREADING".in.move_hp )
   END_RUNG
   RUNG wire#powerrail
      Contact( "FLAGS".STATION.IN_HP_STEP )
   END_RUNG wire#w1
   // the same network as SCL:
   "DBVALVES"."ST3 SWORD A SPREADING".in.move_hp := ("DBVALVES"."ST3 SWORD A SPREADING".test.fp_HP OR "FLAGS".STATION.IN_HP_STEP) AND NOT "FLAGS".STATION.CURTAIN.BREAK;
END_REGION

REGION Network 83: ST3 SWORD A SPREADING WP CLOSE
   // CONDICIONES DE SEGURIDAD / WARUNKI BEZPIECZENSTWA
   RUNG wire#powerrail
      Contact( "DBVALVES"."ST3 SWORD A SPREADING".test.fp_WP )
      I_Contact( "FLAGS".STATION.CURTAIN.BREAK )
      Coil( "DBVALVES"."ST3 SWORD A SPREADING".in.move_wp )
   END_RUNG
   // the same network as SCL:
   "DBVALVES"."ST3 SWORD A SPREADING".in.move_wp := "DBVALVES"."ST3 SWORD A SPREADING".test.fp_WP AND NOT "FLAGS".STATION.CURTAIN.BREAK;
END_REGION

REGION Network 84: SWORD A SPREADING IDLE
   // CONDICIONES DE SEGURIDAD / WARUNKI BEZPIECZENSTWA
   RUNG wire#powerrail
      Contact( "DBVALVES"."ST3 SWORD A SPREADING".test.fp_IDLE )
      wire#w1
      Coil( "DBVALVES"."ST3 SWORD A SPREADING".in.move_idle )
   END_RUNG
   RUNG wire#powerrail
      Contact( "FLAGS".STATION.CURTAIN.BREAK )
   END_RUNG wire#w1
   // the same network as SCL:
   "DBVALVES"."ST3 SWORD A SPREADING".in.move_idle := "DBVALVES"."ST3 SWORD A SPREADING".test.fp_IDLE OR "FLAGS".STATION.CURTAIN.BREAK;
END_REGION

REGION Network 85: ------ [22] ST3 SWORD A OPENING ------
   // SWORD A OPENING
END_REGION

REGION Network 86: ST3 SWORD A OPENING HP OPEN
   // CONDICIONES DE SEGURIDAD / WARUNKI BEZPIECZENSTWA
   RUNG wire#powerrail
      Contact( "DBVALVES"."ST3 SWORD A OPENING".test.fp_HP )
      wire#w1
      I_Contact( "FLAGS".STATION.CURTAIN.BREAK )
      Coil( "DBVALVES"."ST3 SWORD A OPENING".in.move_hp )
   END_RUNG
   RUNG wire#powerrail
      Contact( "FLAGS".STATION.IN_HP_STEP )
   END_RUNG wire#w1
   // the same network as SCL:
   "DBVALVES"."ST3 SWORD A OPENING".in.move_hp := ("DBVALVES"."ST3 SWORD A OPENING".test.fp_HP OR "FLAGS".STATION.IN_HP_STEP) AND NOT "FLAGS".STATION.CURTAIN.BREAK;
END_REGION

REGION Network 87: ST3 SWORD A OPENING WP CLOSE
   // CONDICIONES DE SEGURIDAD / WARUNKI BEZPIECZENSTWA
   RUNG wire#powerrail
      Contact( "DBVALVES"."ST3 SWORD A OPENING".test.fp_WP )
      I_Contact( "FLAGS".STATION.CURTAIN.BREAK )
      Coil( "DBVALVES"."ST3 SWORD A OPENING".in.move_wp )
   END_RUNG
   // the same network as SCL:
   "DBVALVES"."ST3 SWORD A OPENING".in.move_wp := "DBVALVES"."ST3 SWORD A OPENING".test.fp_WP AND NOT "FLAGS".STATION.CURTAIN.BREAK;
END_REGION

REGION Network 88: SWORD A OPENING IDLE
   // CONDICIONES DE SEGURIDAD / WARUNKI BEZPIECZENSTWA
   RUNG wire#powerrail
      Contact( "DBVALVES"."ST3 SWORD A OPENING".test.fp_IDLE )
      wire#w1
      Coil( "DBVALVES"."ST3 SWORD A OPENING".in.move_idle )
   END_RUNG
   RUNG wire#powerrail
      Contact( "FLAGS".STATION.CURTAIN.BREAK )
   END_RUNG wire#w1
   // the same network as SCL:
   "DBVALVES"."ST3 SWORD A OPENING".in.move_idle := "DBVALVES"."ST3 SWORD A OPENING".test.fp_IDLE OR "FLAGS".STATION.CURTAIN.BREAK;
END_REGION

REGION Network 89: ------ [23] ST3 SWORD B SQUEEZING ------
   // SWORD B SQUEEZING
END_REGION

REGION Network 90: ST3 SWORD B SQUEEZING HP OPEN
   // CONDICIONES DE SEGURIDAD / WARUNKI BEZPIECZENSTWA
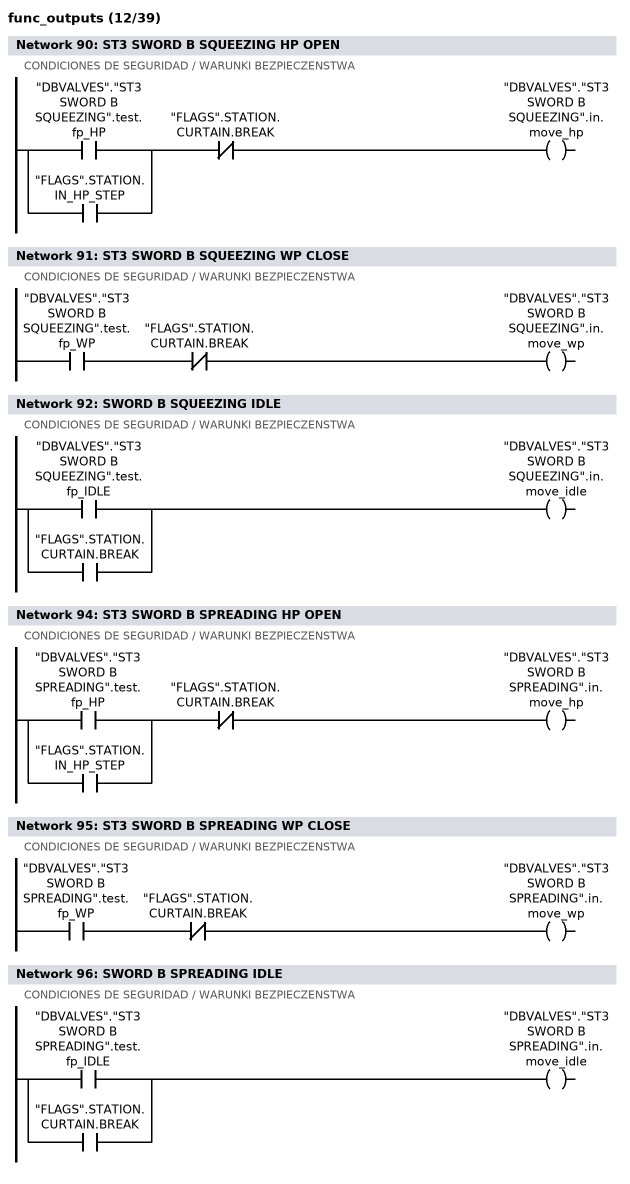
   RUNG wire#powerrail
      Contact( "DBVALVES"."ST3 SWORD B SQUEEZING".test.fp_HP )
      wire#w1
      I_Contact( "FLAGS".STATION.CURTAIN.BREAK )
      Coil( "DBVALVES"."ST3 SWORD B SQUEEZING".in.move_hp )
   END_RUNG
   RUNG wire#powerrail
      Contact( "FLAGS".STATION.IN_HP_STEP )
   END_RUNG wire#w1
   // the same network as SCL:
   "DBVALVES"."ST3 SWORD B SQUEEZING".in.move_hp := ("DBVALVES"."ST3 SWORD B SQUEEZING".test.fp_HP OR "FLAGS".STATION.IN_HP_STEP) AND NOT "FLAGS".STATION.CURTAIN.BREAK;
END_REGION

REGION Network 91: ST3 SWORD B SQUEEZING WP CLOSE
   // CONDICIONES DE SEGURIDAD / WARUNKI BEZPIECZENSTWA
   RUNG wire#powerrail
      Contact( "DBVALVES"."ST3 SWORD B SQUEEZING".test.fp_WP )
      I_Contact( "FLAGS".STATION.CURTAIN.BREAK )
      Coil( "DBVALVES"."ST3 SWORD B SQUEEZING".in.move_wp )
   END_RUNG
   // the same network as SCL:
   "DBVALVES"."ST3 SWORD B SQUEEZING".in.move_wp := "DBVALVES"."ST3 SWORD B SQUEEZING".test.fp_WP AND NOT "FLAGS".STATION.CURTAIN.BREAK;
END_REGION

REGION Network 92: SWORD B SQUEEZING IDLE
   // CONDICIONES DE SEGURIDAD / WARUNKI BEZPIECZENSTWA
   RUNG wire#powerrail
      Contact( "DBVALVES"."ST3 SWORD B SQUEEZING".test.fp_IDLE )
      wire#w1
      Coil( "DBVALVES"."ST3 SWORD B SQUEEZING".in.move_idle )
   END_RUNG
   RUNG wire#powerrail
      Contact( "FLAGS".STATION.CURTAIN.BREAK )
   END_RUNG wire#w1
   // the same network as SCL:
   "DBVALVES"."ST3 SWORD B SQUEEZING".in.move_idle := "DBVALVES"."ST3 SWORD B SQUEEZING".test.fp_IDLE OR "FLAGS".STATION.CURTAIN.BREAK;
END_REGION

REGION Network 93: ------ [24] ST3 SWORD B SPREADING ------
   // SWORD B SPREADING
END_REGION

REGION Network 94: ST3 SWORD B SPREADING HP OPEN
   // CONDICIONES DE SEGURIDAD / WARUNKI BEZPIECZENSTWA
   RUNG wire#powerrail
      Contact( "DBVALVES"."ST3 SWORD B SPREADING".test.fp_HP )
      wire#w1
      I_Contact( "FLAGS".STATION.CURTAIN.BREAK )
      Coil( "DBVALVES"."ST3 SWORD B SPREADING".in.move_hp )
   END_RUNG
   RUNG wire#powerrail
      Contact( "FLAGS".STATION.IN_HP_STEP )
   END_RUNG wire#w1
   // the same network as SCL:
   "DBVALVES"."ST3 SWORD B SPREADING".in.move_hp := ("DBVALVES"."ST3 SWORD B SPREADING".test.fp_HP OR "FLAGS".STATION.IN_HP_STEP) AND NOT "FLAGS".STATION.CURTAIN.BREAK;
END_REGION

REGION Network 95: ST3 SWORD B SPREADING WP CLOSE
   // CONDICIONES DE SEGURIDAD / WARUNKI BEZPIECZENSTWA
   RUNG wire#powerrail
      Contact( "DBVALVES"."ST3 SWORD B SPREADING".test.fp_WP )
      I_Contact( "FLAGS".STATION.CURTAIN.BREAK )
      Coil( "DBVALVES"."ST3 SWORD B SPREADING".in.move_wp )
   END_RUNG
   // the same network as SCL:
   "DBVALVES"."ST3 SWORD B SPREADING".in.move_wp := "DBVALVES"."ST3 SWORD B SPREADING".test.fp_WP AND NOT "FLAGS".STATION.CURTAIN.BREAK;
END_REGION

REGION Network 96: SWORD B SPREADING IDLE
   // CONDICIONES DE SEGURIDAD / WARUNKI BEZPIECZENSTWA
   RUNG wire#powerrail
      Contact( "DBVALVES"."ST3 SWORD B SPREADING".test.fp_IDLE )
      wire#w1
      Coil( "DBVALVES"."ST3 SWORD B SPREADING".in.move_idle )
   END_RUNG
   RUNG wire#powerrail
      Contact( "FLAGS".STATION.CURTAIN.BREAK )
   END_RUNG wire#w1
   // the same network as SCL:
   "DBVALVES"."ST3 SWORD B SPREADING".in.move_idle := "DBVALVES"."ST3 SWORD B SPREADING".test.fp_IDLE OR "FLAGS".STATION.CURTAIN.BREAK;
END_REGION

REGION Network 97: ------ [25] ST3 SWORD B OPENING ------
   // SWORD B OPENING
END_REGION

REGION Network 98: ST3 SWORD B OPENING HP OPEN
   // CONDICIONES DE SEGURIDAD / WARUNKI BEZPIECZENSTWA
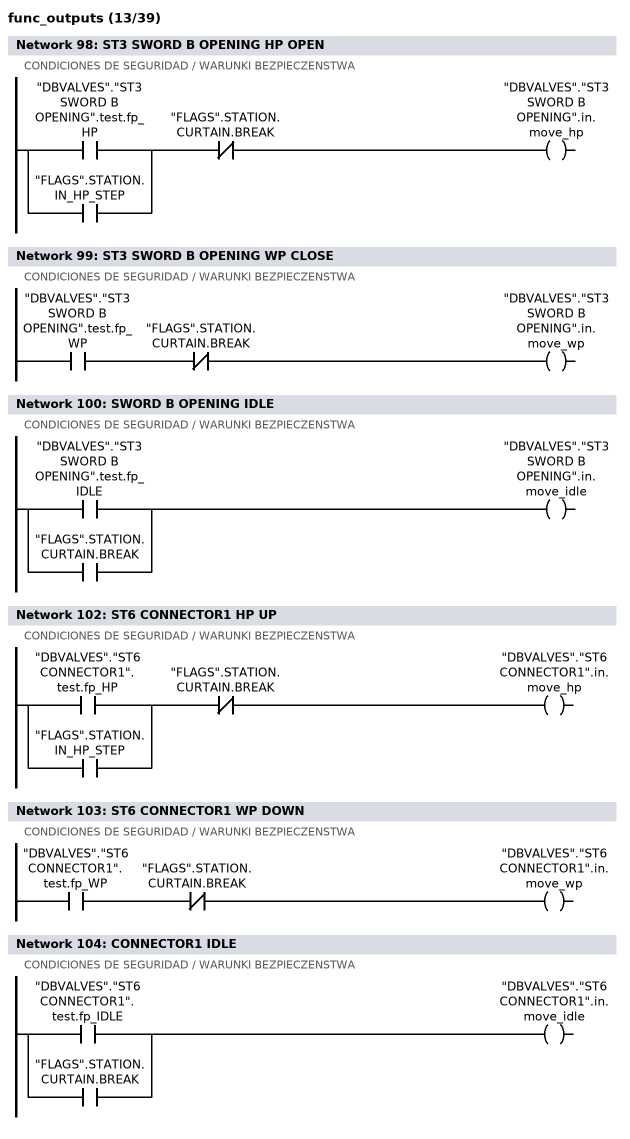
   RUNG wire#powerrail
      Contact( "DBVALVES"."ST3 SWORD B OPENING".test.fp_HP )
      wire#w1
      I_Contact( "FLAGS".STATION.CURTAIN.BREAK )
      Coil( "DBVALVES"."ST3 SWORD B OPENING".in.move_hp )
   END_RUNG
   RUNG wire#powerrail
      Contact( "FLAGS".STATION.IN_HP_STEP )
   END_RUNG wire#w1
   // the same network as SCL:
   "DBVALVES"."ST3 SWORD B OPENING".in.move_hp := ("DBVALVES"."ST3 SWORD B OPENING".test.fp_HP OR "FLAGS".STATION.IN_HP_STEP) AND NOT "FLAGS".STATION.CURTAIN.BREAK;
END_REGION

REGION Network 99: ST3 SWORD B OPENING WP CLOSE
   // CONDICIONES DE SEGURIDAD / WARUNKI BEZPIECZENSTWA
   RUNG wire#powerrail
      Contact( "DBVALVES"."ST3 SWORD B OPENING".test.fp_WP )
      I_Contact( "FLAGS".STATION.CURTAIN.BREAK )
      Coil( "DBVALVES"."ST3 SWORD B OPENING".in.move_wp )
   END_RUNG
   // the same network as SCL:
   "DBVALVES"."ST3 SWORD B OPENING".in.move_wp := "DBVALVES"."ST3 SWORD B OPENING".test.fp_WP AND NOT "FLAGS".STATION.CURTAIN.BREAK;
END_REGION

REGION Network 100: SWORD B OPENING IDLE
   // CONDICIONES DE SEGURIDAD / WARUNKI BEZPIECZENSTWA
   RUNG wire#powerrail
      Contact( "DBVALVES"."ST3 SWORD B OPENING".test.fp_IDLE )
      wire#w1
      Coil( "DBVALVES"."ST3 SWORD B OPENING".in.move_idle )
   END_RUNG
   RUNG wire#powerrail
      Contact( "FLAGS".STATION.CURTAIN.BREAK )
   END_RUNG wire#w1
   // the same network as SCL:
   "DBVALVES"."ST3 SWORD B OPENING".in.move_idle := "DBVALVES"."ST3 SWORD B OPENING".test.fp_IDLE OR "FLAGS".STATION.CURTAIN.BREAK;
END_REGION

REGION Network 101: ------ [26] ST6 CONNECTOR1 ------
   // CONNECTOR1
END_REGION

REGION Network 102: ST6 CONNECTOR1 HP UP
   // CONDICIONES DE SEGURIDAD / WARUNKI BEZPIECZENSTWA
   RUNG wire#powerrail
      Contact( "DBVALVES"."ST6 CONNECTOR1".test.fp_HP )
      wire#w1
      I_Contact( "FLAGS".STATION.CURTAIN.BREAK )
      Coil( "DBVALVES"."ST6 CONNECTOR1".in.move_hp )
   END_RUNG
   RUNG wire#powerrail
      Contact( "FLAGS".STATION.IN_HP_STEP )
   END_RUNG wire#w1
   // the same network as SCL:
   "DBVALVES"."ST6 CONNECTOR1".in.move_hp := ("DBVALVES"."ST6 CONNECTOR1".test.fp_HP OR "FLAGS".STATION.IN_HP_STEP) AND NOT "FLAGS".STATION.CURTAIN.BREAK;
END_REGION

REGION Network 103: ST6 CONNECTOR1 WP DOWN
   // CONDICIONES DE SEGURIDAD / WARUNKI BEZPIECZENSTWA
   RUNG wire#powerrail
      Contact( "DBVALVES"."ST6 CONNECTOR1".test.fp_WP )
      I_Contact( "FLAGS".STATION.CURTAIN.BREAK )
      Coil( "DBVALVES"."ST6 CONNECTOR1".in.move_wp )
   END_RUNG
   // the same network as SCL:
   "DBVALVES"."ST6 CONNECTOR1".in.move_wp := "DBVALVES"."ST6 CONNECTOR1".test.fp_WP AND NOT "FLAGS".STATION.CURTAIN.BREAK;
END_REGION

REGION Network 104: CONNECTOR1 IDLE
   // CONDICIONES DE SEGURIDAD / WARUNKI BEZPIECZENSTWA
   RUNG wire#powerrail
      Contact( "DBVALVES"."ST6 CONNECTOR1".test.fp_IDLE )
      wire#w1
      Coil( "DBVALVES"."ST6 CONNECTOR1".in.move_idle )
   END_RUNG
   RUNG wire#powerrail
      Contact( "FLAGS".STATION.CURTAIN.BREAK )
   END_RUNG wire#w1
   // the same network as SCL:
   "DBVALVES"."ST6 CONNECTOR1".in.move_idle := "DBVALVES"."ST6 CONNECTOR1".test.fp_IDLE OR "FLAGS".STATION.CURTAIN.BREAK;
END_REGION

REGION Network 105: ------ [27] ST6 CONNECTOR2 ------
   // CONNECTOR2
END_REGION

REGION Network 106: ST6 CONNECTOR2 HP UP
   // CONDICIONES DE SEGURIDAD / WARUNKI BEZPIECZENSTWA
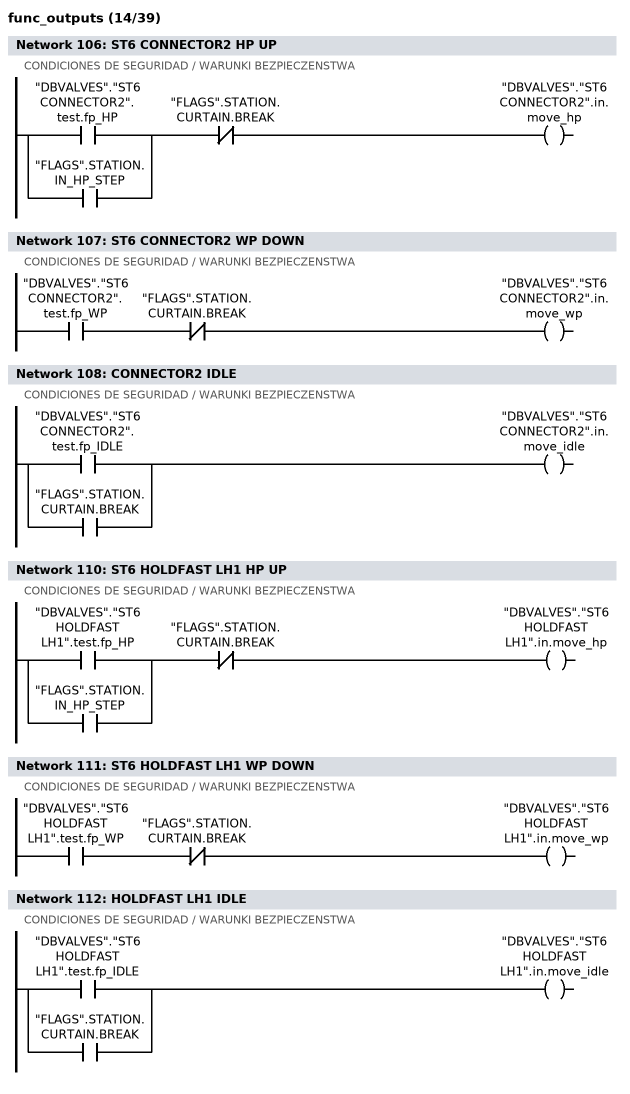
   RUNG wire#powerrail
      Contact( "DBVALVES"."ST6 CONNECTOR2".test.fp_HP )
      wire#w1
      I_Contact( "FLAGS".STATION.CURTAIN.BREAK )
      Coil( "DBVALVES"."ST6 CONNECTOR2".in.move_hp )
   END_RUNG
   RUNG wire#powerrail
      Contact( "FLAGS".STATION.IN_HP_STEP )
   END_RUNG wire#w1
   // the same network as SCL:
   "DBVALVES"."ST6 CONNECTOR2".in.move_hp := ("DBVALVES"."ST6 CONNECTOR2".test.fp_HP OR "FLAGS".STATION.IN_HP_STEP) AND NOT "FLAGS".STATION.CURTAIN.BREAK;
END_REGION

REGION Network 107: ST6 CONNECTOR2 WP DOWN
   // CONDICIONES DE SEGURIDAD / WARUNKI BEZPIECZENSTWA
   RUNG wire#powerrail
      Contact( "DBVALVES"."ST6 CONNECTOR2".test.fp_WP )
      I_Contact( "FLAGS".STATION.CURTAIN.BREAK )
      Coil( "DBVALVES"."ST6 CONNECTOR2".in.move_wp )
   END_RUNG
   // the same network as SCL:
   "DBVALVES"."ST6 CONNECTOR2".in.move_wp := "DBVALVES"."ST6 CONNECTOR2".test.fp_WP AND NOT "FLAGS".STATION.CURTAIN.BREAK;
END_REGION

REGION Network 108: CONNECTOR2 IDLE
   // CONDICIONES DE SEGURIDAD / WARUNKI BEZPIECZENSTWA
   RUNG wire#powerrail
      Contact( "DBVALVES"."ST6 CONNECTOR2".test.fp_IDLE )
      wire#w1
      Coil( "DBVALVES"."ST6 CONNECTOR2".in.move_idle )
   END_RUNG
   RUNG wire#powerrail
      Contact( "FLAGS".STATION.CURTAIN.BREAK )
   END_RUNG wire#w1
   // the same network as SCL:
   "DBVALVES"."ST6 CONNECTOR2".in.move_idle := "DBVALVES"."ST6 CONNECTOR2".test.fp_IDLE OR "FLAGS".STATION.CURTAIN.BREAK;
END_REGION

REGION Network 109: ------ [28] ST6 HOLDFAST LH1 ------
   // HOLDFAST LH1
END_REGION

REGION Network 110: ST6 HOLDFAST LH1 HP UP
   // CONDICIONES DE SEGURIDAD / WARUNKI BEZPIECZENSTWA
   RUNG wire#powerrail
      Contact( "DBVALVES"."ST6 HOLDFAST LH1".test.fp_HP )
      wire#w1
      I_Contact( "FLAGS".STATION.CURTAIN.BREAK )
      Coil( "DBVALVES"."ST6 HOLDFAST LH1".in.move_hp )
   END_RUNG
   RUNG wire#powerrail
      Contact( "FLAGS".STATION.IN_HP_STEP )
   END_RUNG wire#w1
   // the same network as SCL:
   "DBVALVES"."ST6 HOLDFAST LH1".in.move_hp := ("DBVALVES"."ST6 HOLDFAST LH1".test.fp_HP OR "FLAGS".STATION.IN_HP_STEP) AND NOT "FLAGS".STATION.CURTAIN.BREAK;
END_REGION

REGION Network 111: ST6 HOLDFAST LH1 WP DOWN
   // CONDICIONES DE SEGURIDAD / WARUNKI BEZPIECZENSTWA
   RUNG wire#powerrail
      Contact( "DBVALVES"."ST6 HOLDFAST LH1".test.fp_WP )
      I_Contact( "FLAGS".STATION.CURTAIN.BREAK )
      Coil( "DBVALVES"."ST6 HOLDFAST LH1".in.move_wp )
   END_RUNG
   // the same network as SCL:
   "DBVALVES"."ST6 HOLDFAST LH1".in.move_wp := "DBVALVES"."ST6 HOLDFAST LH1".test.fp_WP AND NOT "FLAGS".STATION.CURTAIN.BREAK;
END_REGION

REGION Network 112: HOLDFAST LH1 IDLE
   // CONDICIONES DE SEGURIDAD / WARUNKI BEZPIECZENSTWA
   RUNG wire#powerrail
      Contact( "DBVALVES"."ST6 HOLDFAST LH1".test.fp_IDLE )
      wire#w1
      Coil( "DBVALVES"."ST6 HOLDFAST LH1".in.move_idle )
   END_RUNG
   RUNG wire#powerrail
      Contact( "FLAGS".STATION.CURTAIN.BREAK )
   END_RUNG wire#w1
   // the same network as SCL:
   "DBVALVES"."ST6 HOLDFAST LH1".in.move_idle := "DBVALVES"."ST6 HOLDFAST LH1".test.fp_IDLE OR "FLAGS".STATION.CURTAIN.BREAK;
END_REGION

REGION Network 113: ------ [29] ST6 HOLDFAST LH2 ------
   // HOLDFAST LH2
END_REGION

REGION Network 114: ST6 HOLDFAST LH2 HP UP
   // CONDICIONES DE SEGURIDAD / WARUNKI BEZPIECZENSTWA
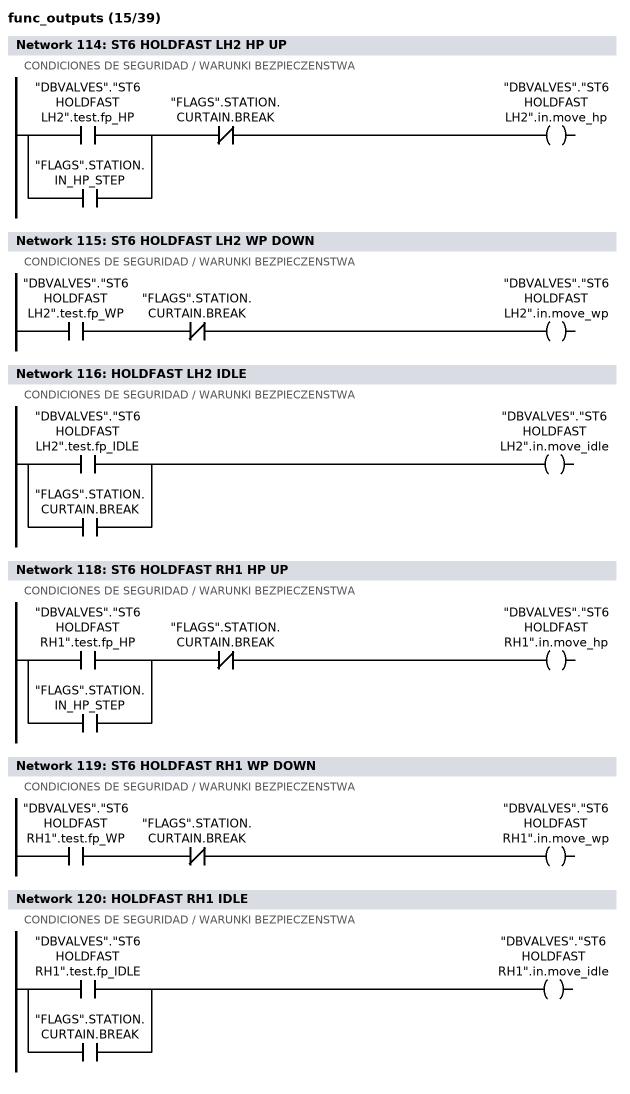
   RUNG wire#powerrail
      Contact( "DBVALVES"."ST6 HOLDFAST LH2".test.fp_HP )
      wire#w1
      I_Contact( "FLAGS".STATION.CURTAIN.BREAK )
      Coil( "DBVALVES"."ST6 HOLDFAST LH2".in.move_hp )
   END_RUNG
   RUNG wire#powerrail
      Contact( "FLAGS".STATION.IN_HP_STEP )
   END_RUNG wire#w1
   // the same network as SCL:
   "DBVALVES"."ST6 HOLDFAST LH2".in.move_hp := ("DBVALVES"."ST6 HOLDFAST LH2".test.fp_HP OR "FLAGS".STATION.IN_HP_STEP) AND NOT "FLAGS".STATION.CURTAIN.BREAK;
END_REGION

REGION Network 115: ST6 HOLDFAST LH2 WP DOWN
   // CONDICIONES DE SEGURIDAD / WARUNKI BEZPIECZENSTWA
   RUNG wire#powerrail
      Contact( "DBVALVES"."ST6 HOLDFAST LH2".test.fp_WP )
      I_Contact( "FLAGS".STATION.CURTAIN.BREAK )
      Coil( "DBVALVES"."ST6 HOLDFAST LH2".in.move_wp )
   END_RUNG
   // the same network as SCL:
   "DBVALVES"."ST6 HOLDFAST LH2".in.move_wp := "DBVALVES"."ST6 HOLDFAST LH2".test.fp_WP AND NOT "FLAGS".STATION.CURTAIN.BREAK;
END_REGION

REGION Network 116: HOLDFAST LH2 IDLE
   // CONDICIONES DE SEGURIDAD / WARUNKI BEZPIECZENSTWA
   RUNG wire#powerrail
      Contact( "DBVALVES"."ST6 HOLDFAST LH2".test.fp_IDLE )
      wire#w1
      Coil( "DBVALVES"."ST6 HOLDFAST LH2".in.move_idle )
   END_RUNG
   RUNG wire#powerrail
      Contact( "FLAGS".STATION.CURTAIN.BREAK )
   END_RUNG wire#w1
   // the same network as SCL:
   "DBVALVES"."ST6 HOLDFAST LH2".in.move_idle := "DBVALVES"."ST6 HOLDFAST LH2".test.fp_IDLE OR "FLAGS".STATION.CURTAIN.BREAK;
END_REGION

REGION Network 117: ------ [30] ST6 HOLDFAST RH1 ------
   // HOLDFAST RH1
END_REGION

REGION Network 118: ST6 HOLDFAST RH1 HP UP
   // CONDICIONES DE SEGURIDAD / WARUNKI BEZPIECZENSTWA
   RUNG wire#powerrail
      Contact( "DBVALVES"."ST6 HOLDFAST RH1".test.fp_HP )
      wire#w1
      I_Contact( "FLAGS".STATION.CURTAIN.BREAK )
      Coil( "DBVALVES"."ST6 HOLDFAST RH1".in.move_hp )
   END_RUNG
   RUNG wire#powerrail
      Contact( "FLAGS".STATION.IN_HP_STEP )
   END_RUNG wire#w1
   // the same network as SCL:
   "DBVALVES"."ST6 HOLDFAST RH1".in.move_hp := ("DBVALVES"."ST6 HOLDFAST RH1".test.fp_HP OR "FLAGS".STATION.IN_HP_STEP) AND NOT "FLAGS".STATION.CURTAIN.BREAK;
END_REGION

REGION Network 119: ST6 HOLDFAST RH1 WP DOWN
   // CONDICIONES DE SEGURIDAD / WARUNKI BEZPIECZENSTWA
   RUNG wire#powerrail
      Contact( "DBVALVES"."ST6 HOLDFAST RH1".test.fp_WP )
      I_Contact( "FLAGS".STATION.CURTAIN.BREAK )
      Coil( "DBVALVES"."ST6 HOLDFAST RH1".in.move_wp )
   END_RUNG
   // the same network as SCL:
   "DBVALVES"."ST6 HOLDFAST RH1".in.move_wp := "DBVALVES"."ST6 HOLDFAST RH1".test.fp_WP AND NOT "FLAGS".STATION.CURTAIN.BREAK;
END_REGION

REGION Network 120: HOLDFAST RH1 IDLE
   // CONDICIONES DE SEGURIDAD / WARUNKI BEZPIECZENSTWA
   RUNG wire#powerrail
      Contact( "DBVALVES"."ST6 HOLDFAST RH1".test.fp_IDLE )
      wire#w1
      Coil( "DBVALVES"."ST6 HOLDFAST RH1".in.move_idle )
   END_RUNG
   RUNG wire#powerrail
      Contact( "FLAGS".STATION.CURTAIN.BREAK )
   END_RUNG wire#w1
   // the same network as SCL:
   "DBVALVES"."ST6 HOLDFAST RH1".in.move_idle := "DBVALVES"."ST6 HOLDFAST RH1".test.fp_IDLE OR "FLAGS".STATION.CURTAIN.BREAK;
END_REGION

REGION Network 121: ------ [31] ST6 HOLDFAST RH2 ------
   // HOLDFAST RH2
END_REGION

REGION Network 122: ST6 HOLDFAST RH2 HP UP
   // CONDICIONES DE SEGURIDAD / WARUNKI BEZPIECZENSTWA
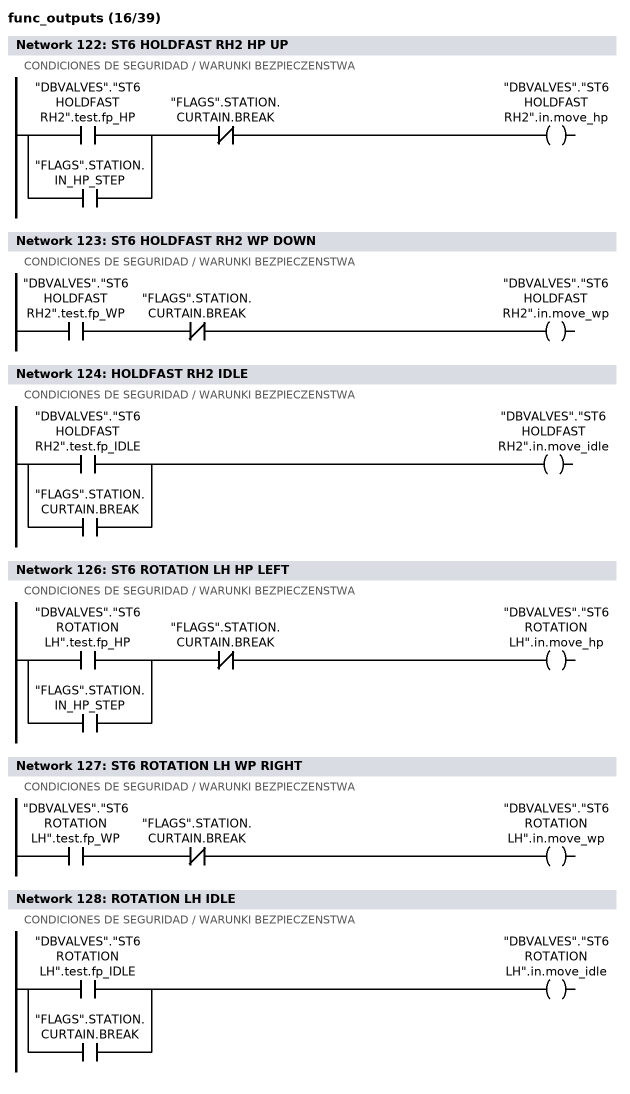
   RUNG wire#powerrail
      Contact( "DBVALVES"."ST6 HOLDFAST RH2".test.fp_HP )
      wire#w1
      I_Contact( "FLAGS".STATION.CURTAIN.BREAK )
      Coil( "DBVALVES"."ST6 HOLDFAST RH2".in.move_hp )
   END_RUNG
   RUNG wire#powerrail
      Contact( "FLAGS".STATION.IN_HP_STEP )
   END_RUNG wire#w1
   // the same network as SCL:
   "DBVALVES"."ST6 HOLDFAST RH2".in.move_hp := ("DBVALVES"."ST6 HOLDFAST RH2".test.fp_HP OR "FLAGS".STATION.IN_HP_STEP) AND NOT "FLAGS".STATION.CURTAIN.BREAK;
END_REGION

REGION Network 123: ST6 HOLDFAST RH2 WP DOWN
   // CONDICIONES DE SEGURIDAD / WARUNKI BEZPIECZENSTWA
   RUNG wire#powerrail
      Contact( "DBVALVES"."ST6 HOLDFAST RH2".test.fp_WP )
      I_Contact( "FLAGS".STATION.CURTAIN.BREAK )
      Coil( "DBVALVES"."ST6 HOLDFAST RH2".in.move_wp )
   END_RUNG
   // the same network as SCL:
   "DBVALVES"."ST6 HOLDFAST RH2".in.move_wp := "DBVALVES"."ST6 HOLDFAST RH2".test.fp_WP AND NOT "FLAGS".STATION.CURTAIN.BREAK;
END_REGION

REGION Network 124: HOLDFAST RH2 IDLE
   // CONDICIONES DE SEGURIDAD / WARUNKI BEZPIECZENSTWA
   RUNG wire#powerrail
      Contact( "DBVALVES"."ST6 HOLDFAST RH2".test.fp_IDLE )
      wire#w1
      Coil( "DBVALVES"."ST6 HOLDFAST RH2".in.move_idle )
   END_RUNG
   RUNG wire#powerrail
      Contact( "FLAGS".STATION.CURTAIN.BREAK )
   END_RUNG wire#w1
   // the same network as SCL:
   "DBVALVES"."ST6 HOLDFAST RH2".in.move_idle := "DBVALVES"."ST6 HOLDFAST RH2".test.fp_IDLE OR "FLAGS".STATION.CURTAIN.BREAK;
END_REGION

REGION Network 125: ------ [32] ST6 ROTATION LH ------
   // ROTATION LH
END_REGION

REGION Network 126: ST6 ROTATION LH HP LEFT
   // CONDICIONES DE SEGURIDAD / WARUNKI BEZPIECZENSTWA
   RUNG wire#powerrail
      Contact( "DBVALVES"."ST6 ROTATION LH".test.fp_HP )
      wire#w1
      I_Contact( "FLAGS".STATION.CURTAIN.BREAK )
      Coil( "DBVALVES"."ST6 ROTATION LH".in.move_hp )
   END_RUNG
   RUNG wire#powerrail
      Contact( "FLAGS".STATION.IN_HP_STEP )
   END_RUNG wire#w1
   // the same network as SCL:
   "DBVALVES"."ST6 ROTATION LH".in.move_hp := ("DBVALVES"."ST6 ROTATION LH".test.fp_HP OR "FLAGS".STATION.IN_HP_STEP) AND NOT "FLAGS".STATION.CURTAIN.BREAK;
END_REGION

REGION Network 127: ST6 ROTATION LH WP RIGHT
   // CONDICIONES DE SEGURIDAD / WARUNKI BEZPIECZENSTWA
   RUNG wire#powerrail
      Contact( "DBVALVES"."ST6 ROTATION LH".test.fp_WP )
      I_Contact( "FLAGS".STATION.CURTAIN.BREAK )
      Coil( "DBVALVES"."ST6 ROTATION LH".in.move_wp )
   END_RUNG
   // the same network as SCL:
   "DBVALVES"."ST6 ROTATION LH".in.move_wp := "DBVALVES"."ST6 ROTATION LH".test.fp_WP AND NOT "FLAGS".STATION.CURTAIN.BREAK;
END_REGION

REGION Network 128: ROTATION LH IDLE
   // CONDICIONES DE SEGURIDAD / WARUNKI BEZPIECZENSTWA
   RUNG wire#powerrail
      Contact( "DBVALVES"."ST6 ROTATION LH".test.fp_IDLE )
      wire#w1
      Coil( "DBVALVES"."ST6 ROTATION LH".in.move_idle )
   END_RUNG
   RUNG wire#powerrail
      Contact( "FLAGS".STATION.CURTAIN.BREAK )
   END_RUNG wire#w1
   // the same network as SCL:
   "DBVALVES"."ST6 ROTATION LH".in.move_idle := "DBVALVES"."ST6 ROTATION LH".test.fp_IDLE OR "FLAGS".STATION.CURTAIN.BREAK;
END_REGION

REGION Network 129: ------ [33] ST6 ROTATION RH ------
   // ROTATION RH
END_REGION

REGION Network 130: ST6 ROTATION RH HP RIGHT
   // CONDICIONES DE SEGURIDAD / WARUNKI BEZPIECZENSTWA
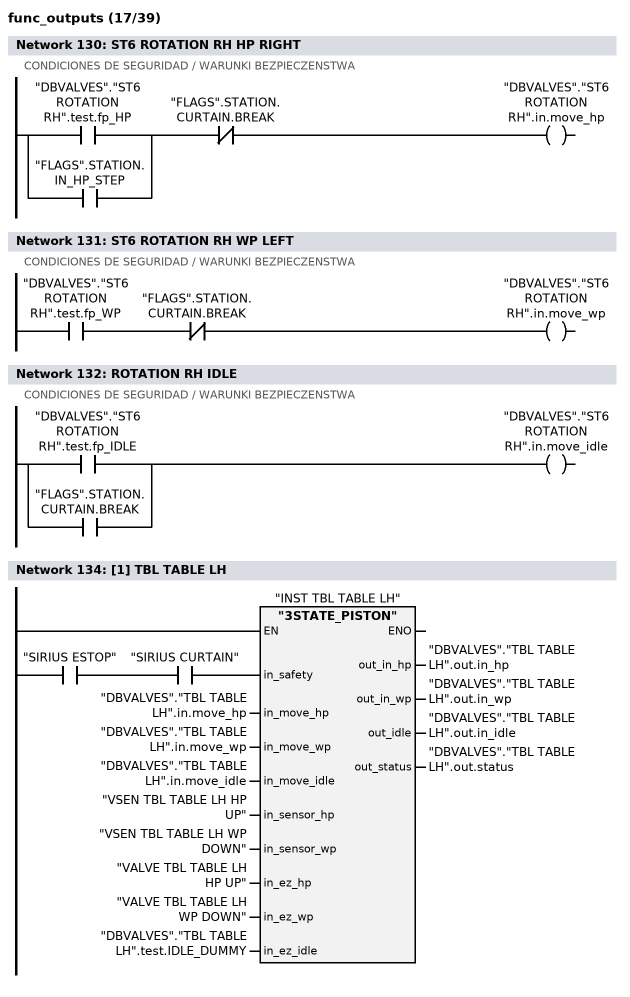
   RUNG wire#powerrail
      Contact( "DBVALVES"."ST6 ROTATION RH".test.fp_HP )
      wire#w1
      I_Contact( "FLAGS".STATION.CURTAIN.BREAK )
      Coil( "DBVALVES"."ST6 ROTATION RH".in.move_hp )
   END_RUNG
   RUNG wire#powerrail
      Contact( "FLAGS".STATION.IN_HP_STEP )
   END_RUNG wire#w1
   // the same network as SCL:
   "DBVALVES"."ST6 ROTATION RH".in.move_hp := ("DBVALVES"."ST6 ROTATION RH".test.fp_HP OR "FLAGS".STATION.IN_HP_STEP) AND NOT "FLAGS".STATION.CURTAIN.BREAK;
END_REGION

REGION Network 131: ST6 ROTATION RH WP LEFT
   // CONDICIONES DE SEGURIDAD / WARUNKI BEZPIECZENSTWA
   RUNG wire#powerrail
      Contact( "DBVALVES"."ST6 ROTATION RH".test.fp_WP )
      I_Contact( "FLAGS".STATION.CURTAIN.BREAK )
      Coil( "DBVALVES"."ST6 ROTATION RH".in.move_wp )
   END_RUNG
   // the same network as SCL:
   "DBVALVES"."ST6 ROTATION RH".in.move_wp := "DBVALVES"."ST6 ROTATION RH".test.fp_WP AND NOT "FLAGS".STATION.CURTAIN.BREAK;
END_REGION

REGION Network 132: ROTATION RH IDLE
   // CONDICIONES DE SEGURIDAD / WARUNKI BEZPIECZENSTWA
   RUNG wire#powerrail
      Contact( "DBVALVES"."ST6 ROTATION RH".test.fp_IDLE )
      wire#w1
      Coil( "DBVALVES"."ST6 ROTATION RH".in.move_idle )
   END_RUNG
   RUNG wire#powerrail
      Contact( "FLAGS".STATION.CURTAIN.BREAK )
   END_RUNG wire#w1
   // the same network as SCL:
   "DBVALVES"."ST6 ROTATION RH".in.move_idle := "DBVALVES"."ST6 ROTATION RH".test.fp_IDLE OR "FLAGS".STATION.CURTAIN.BREAK;
END_REGION

REGION Network 133: ======= VALVES =======
END_REGION

REGION Network 134: [1] TBL TABLE LH
   RUNG wire#powerrail
      "INST TBL TABLE LH"(in_safety := wire#w1, in_move_hp := "DBVALVES"."TBL TABLE LH".in.move_hp, in_move_wp := "DBVALVES"."TBL TABLE LH".in.move_wp, in_move_idle := "DBVALVES"."TBL TABLE LH".in.move_idle, in_sensor_hp := "VSEN TBL TABLE LH HP UP", in_sensor_wp := "VSEN TBL TABLE LH WP DOWN", in_ez_hp := "VALVE TBL TABLE LH HP UP", in_ez_wp := "VALVE TBL TABLE LH WP DOWN", in_ez_idle := "DBVALVES"."TBL TABLE LH".test.IDLE_DUMMY, out_in_hp => "DBVALVES"."TBL TABLE LH".out.in_hp, out_in_wp => "DBVALVES"."TBL TABLE LH".out.in_wp, out_idle => "DBVALVES"."TBL TABLE LH".out.in_idle, out_status => "DBVALVES"."TBL TABLE LH".out.status)
   END_RUNG
   RUNG wire#powerrail
      Contact( "SIRIUS ESTOP" )
      Contact( "SIRIUS CURTAIN" )
   END_RUNG wire#w1
   // the same network as SCL:
   "INST TBL TABLE LH"(in_safety := "SIRIUS ESTOP" AND "SIRIUS CURTAIN",   // "3STATE_PISTON"
                       in_move_hp := "DBVALVES"."TBL TABLE LH".in.move_hp,
                       in_move_wp := "DBVALVES"."TBL TABLE LH".in.move_wp,
                       in_move_idle := "DBVALVES"."TBL TABLE LH".in.move_idle,
                       in_sensor_hp := "VSEN TBL TABLE LH HP UP",
                       in_sensor_wp := "VSEN TBL TABLE LH WP DOWN",
                       in_ez_hp := "VALVE TBL TABLE LH HP UP",
                       in_ez_wp := "VALVE TBL TABLE LH WP DOWN",
                       in_ez_idle := "DBVALVES"."TBL TABLE LH".test.IDLE_DUMMY,
                       out_in_hp => "DBVALVES"."TBL TABLE LH".out.in_hp,
                       out_in_wp => "DBVALVES"."TBL TABLE LH".out.in_wp,
                       out_idle => "DBVALVES"."TBL TABLE LH".out.in_idle,
                       out_status => "DBVALVES"."TBL TABLE LH".out.status);
END_REGION

REGION Network 135: [2] TBL TABLE RH
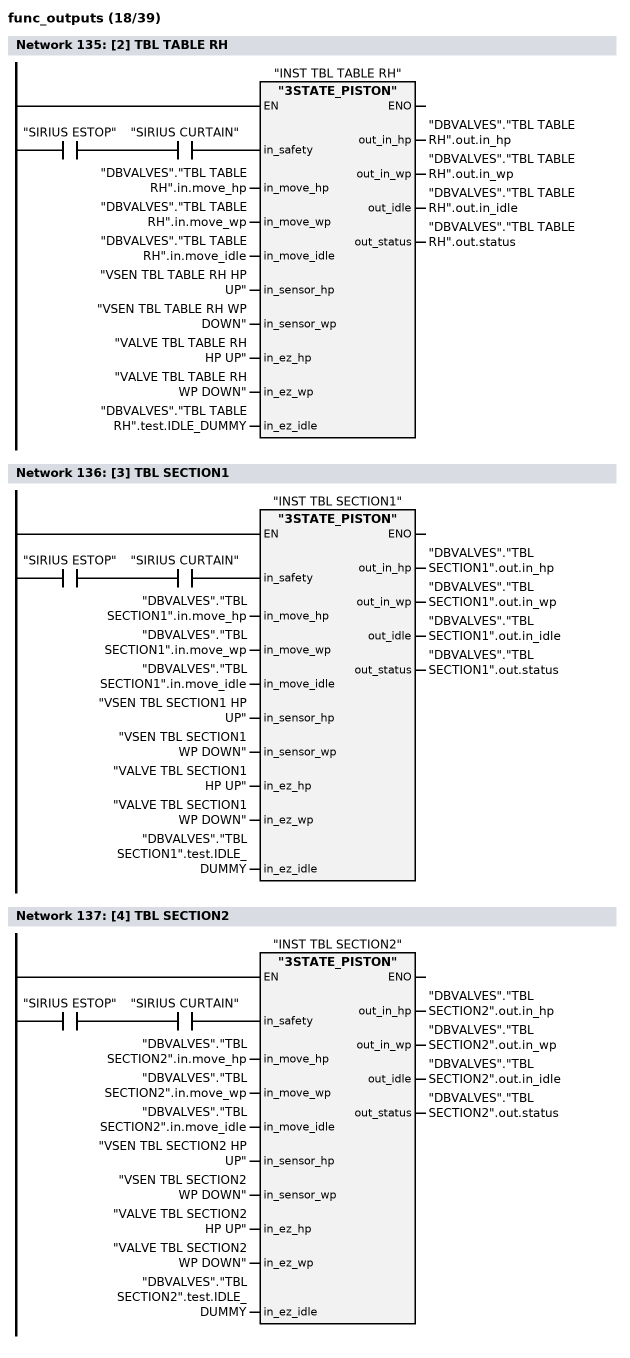
   RUNG wire#powerrail
      "INST TBL TABLE RH"(in_safety := wire#w1, in_move_hp := "DBVALVES"."TBL TABLE RH".in.move_hp, in_move_wp := "DBVALVES"."TBL TABLE RH".in.move_wp, in_move_idle := "DBVALVES"."TBL TABLE RH".in.move_idle, in_sensor_hp := "VSEN TBL TABLE RH HP UP", in_sensor_wp := "VSEN TBL TABLE RH WP DOWN", in_ez_hp := "VALVE TBL TABLE RH HP UP", in_ez_wp := "VALVE TBL TABLE RH WP DOWN", in_ez_idle := "DBVALVES"."TBL TABLE RH".test.IDLE_DUMMY, out_in_hp => "DBVALVES"."TBL TABLE RH".out.in_hp, out_in_wp => "DBVALVES"."TBL TABLE RH".out.in_wp, out_idle => "DBVALVES"."TBL TABLE RH".out.in_idle, out_status => "DBVALVES"."TBL TABLE RH".out.status)
   END_RUNG
   RUNG wire#powerrail
      Contact( "SIRIUS ESTOP" )
      Contact( "SIRIUS CURTAIN" )
   END_RUNG wire#w1
   // the same network as SCL:
   "INST TBL TABLE RH"(in_safety := "SIRIUS ESTOP" AND "SIRIUS CURTAIN",   // "3STATE_PISTON"
                       in_move_hp := "DBVALVES"."TBL TABLE RH".in.move_hp,
                       in_move_wp := "DBVALVES"."TBL TABLE RH".in.move_wp,
                       in_move_idle := "DBVALVES"."TBL TABLE RH".in.move_idle,
                       in_sensor_hp := "VSEN TBL TABLE RH HP UP",
                       in_sensor_wp := "VSEN TBL TABLE RH WP DOWN",
                       in_ez_hp := "VALVE TBL TABLE RH HP UP",
                       in_ez_wp := "VALVE TBL TABLE RH WP DOWN",
                       in_ez_idle := "DBVALVES"."TBL TABLE RH".test.IDLE_DUMMY,
                       out_in_hp => "DBVALVES"."TBL TABLE RH".out.in_hp,
                       out_in_wp => "DBVALVES"."TBL TABLE RH".out.in_wp,
                       out_idle => "DBVALVES"."TBL TABLE RH".out.in_idle,
                       out_status => "DBVALVES"."TBL TABLE RH".out.status);
END_REGION

REGION Network 136: [3] TBL SECTION1
   RUNG wire#powerrail
      "INST TBL SECTION1"(in_safety := wire#w1, in_move_hp := "DBVALVES"."TBL SECTION1".in.move_hp, in_move_wp := "DBVALVES"."TBL SECTION1".in.move_wp, in_move_idle := "DBVALVES"."TBL SECTION1".in.move_idle, in_sensor_hp := "VSEN TBL SECTION1 HP UP", in_sensor_wp := "VSEN TBL SECTION1 WP DOWN", in_ez_hp := "VALVE TBL SECTION1 HP UP", in_ez_wp := "VALVE TBL SECTION1 WP DOWN", in_ez_idle := "DBVALVES"."TBL SECTION1".test.IDLE_DUMMY, out_in_hp => "DBVALVES"."TBL SECTION1".out.in_hp, out_in_wp => "DBVALVES"."TBL SECTION1".out.in_wp, out_idle => "DBVALVES"."TBL SECTION1".out.in_idle, out_status => "DBVALVES"."TBL SECTION1".out.status)
   END_RUNG
   RUNG wire#powerrail
      Contact( "SIRIUS ESTOP" )
      Contact( "SIRIUS CURTAIN" )
   END_RUNG wire#w1
   // the same network as SCL:
   "INST TBL SECTION1"(in_safety := "SIRIUS ESTOP" AND "SIRIUS CURTAIN",   // "3STATE_PISTON"
                       in_move_hp := "DBVALVES"."TBL SECTION1".in.move_hp,
                       in_move_wp := "DBVALVES"."TBL SECTION1".in.move_wp,
                       in_move_idle := "DBVALVES"."TBL SECTION1".in.move_idle,
                       in_sensor_hp := "VSEN TBL SECTION1 HP UP",
                       in_sensor_wp := "VSEN TBL SECTION1 WP DOWN",
                       in_ez_hp := "VALVE TBL SECTION1 HP UP",
                       in_ez_wp := "VALVE TBL SECTION1 WP DOWN",
                       in_ez_idle := "DBVALVES"."TBL SECTION1".test.IDLE_DUMMY,
                       out_in_hp => "DBVALVES"."TBL SECTION1".out.in_hp,
                       out_in_wp => "DBVALVES"."TBL SECTION1".out.in_wp,
                       out_idle => "DBVALVES"."TBL SECTION1".out.in_idle,
                       out_status => "DBVALVES"."TBL SECTION1".out.status);
END_REGION

REGION Network 137: [4] TBL SECTION2
   RUNG wire#powerrail
      "INST TBL SECTION2"(in_safety := wire#w1, in_move_hp := "DBVALVES"."TBL SECTION2".in.move_hp, in_move_wp := "DBVALVES"."TBL SECTION2".in.move_wp, in_move_idle := "DBVALVES"."TBL SECTION2".in.move_idle, in_sensor_hp := "VSEN TBL SECTION2 HP UP", in_sensor_wp := "VSEN TBL SECTION2 WP DOWN", in_ez_hp := "VALVE TBL SECTION2 HP UP", in_ez_wp := "VALVE TBL SECTION2 WP DOWN", in_ez_idle := "DBVALVES"."TBL SECTION2".test.IDLE_DUMMY, out_in_hp => "DBVALVES"."TBL SECTION2".out.in_hp, out_in_wp => "DBVALVES"."TBL SECTION2".out.in_wp, out_idle => "DBVALVES"."TBL SECTION2".out.in_idle, out_status => "DBVALVES"."TBL SECTION2".out.status)
   END_RUNG
   RUNG wire#powerrail
      Contact( "SIRIUS ESTOP" )
      Contact( "SIRIUS CURTAIN" )
   END_RUNG wire#w1
   // the same network as SCL:
   "INST TBL SECTION2"(in_safety := "SIRIUS ESTOP" AND "SIRIUS CURTAIN",   // "3STATE_PISTON"
                       in_move_hp := "DBVALVES"."TBL SECTION2".in.move_hp,
                       in_move_wp := "DBVALVES"."TBL SECTION2".in.move_wp,
                       in_move_idle := "DBVALVES"."TBL SECTION2".in.move_idle,
                       in_sensor_hp := "VSEN TBL SECTION2 HP UP",
                       in_sensor_wp := "VSEN TBL SECTION2 WP DOWN",
                       in_ez_hp := "VALVE TBL SECTION2 HP UP",
                       in_ez_wp := "VALVE TBL SECTION2 WP DOWN",
                       in_ez_idle := "DBVALVES"."TBL SECTION2".test.IDLE_DUMMY,
                       out_in_hp => "DBVALVES"."TBL SECTION2".out.in_hp,
                       out_in_wp => "DBVALVES"."TBL SECTION2".out.in_wp,
                       out_idle => "DBVALVES"."TBL SECTION2".out.in_idle,
                       out_status => "DBVALVES"."TBL SECTION2".out.status);
END_REGION

REGION Network 138: [5] TBL SECTION4 LH
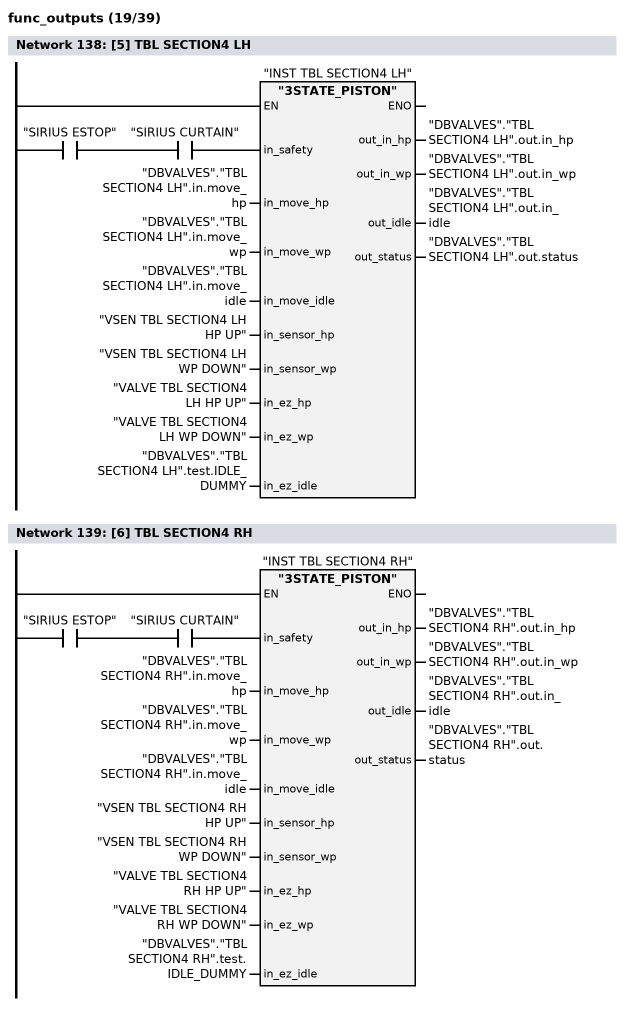
   RUNG wire#powerrail
      "INST TBL SECTION4 LH"(in_safety := wire#w1, in_move_hp := "DBVALVES"."TBL SECTION4 LH".in.move_hp, in_move_wp := "DBVALVES"."TBL SECTION4 LH".in.move_wp, in_move_idle := "DBVALVES"."TBL SECTION4 LH".in.move_idle, in_sensor_hp := "VSEN TBL SECTION4 LH HP UP", in_sensor_wp := "VSEN TBL SECTION4 LH WP DOWN", in_ez_hp := "VALVE TBL SECTION4 LH HP UP", in_ez_wp := "VALVE TBL SECTION4 LH WP DOWN", in_ez_idle := "DBVALVES"."TBL SECTION4 LH".test.IDLE_DUMMY, out_in_hp => "DBVALVES"."TBL SECTION4 LH".out.in_hp, out_in_wp => "DBVALVES"."TBL SECTION4 LH".out.in_wp, out_idle => "DBVALVES"."TBL SECTION4 LH".out.in_idle, out_status => "DBVALVES"."TBL SECTION4 LH".out.status)
   END_RUNG
   RUNG wire#powerrail
      Contact( "SIRIUS ESTOP" )
      Contact( "SIRIUS CURTAIN" )
   END_RUNG wire#w1
   // the same network as SCL:
   "INST TBL SECTION4 LH"(in_safety := "SIRIUS ESTOP" AND "SIRIUS CURTAIN",   // "3STATE_PISTON"
                          in_move_hp := "DBVALVES"."TBL SECTION4 LH".in.move_hp,
                          in_move_wp := "DBVALVES"."TBL SECTION4 LH".in.move_wp,
                          in_move_idle := "DBVALVES"."TBL SECTION4 LH".in.move_idle,
                          in_sensor_hp := "VSEN TBL SECTION4 LH HP UP",
                          in_sensor_wp := "VSEN TBL SECTION4 LH WP DOWN",
                          in_ez_hp := "VALVE TBL SECTION4 LH HP UP",
                          in_ez_wp := "VALVE TBL SECTION4 LH WP DOWN",
                          in_ez_idle := "DBVALVES"."TBL SECTION4 LH".test.IDLE_DUMMY,
                          out_in_hp => "DBVALVES"."TBL SECTION4 LH".out.in_hp,
                          out_in_wp => "DBVALVES"."TBL SECTION4 LH".out.in_wp,
                          out_idle => "DBVALVES"."TBL SECTION4 LH".out.in_idle,
                          out_status => "DBVALVES"."TBL SECTION4 LH".out.status);
END_REGION

REGION Network 139: [6] TBL SECTION4 RH
   RUNG wire#powerrail
      "INST TBL SECTION4 RH"(in_safety := wire#w1, in_move_hp := "DBVALVES"."TBL SECTION4 RH".in.move_hp, in_move_wp := "DBVALVES"."TBL SECTION4 RH".in.move_wp, in_move_idle := "DBVALVES"."TBL SECTION4 RH".in.move_idle, in_sensor_hp := "VSEN TBL SECTION4 RH HP UP", in_sensor_wp := "VSEN TBL SECTION4 RH WP DOWN", in_ez_hp := "VALVE TBL SECTION4 RH HP UP", in_ez_wp := "VALVE TBL SECTION4 RH WP DOWN", in_ez_idle := "DBVALVES"."TBL SECTION4 RH".test.IDLE_DUMMY, out_in_hp => "DBVALVES"."TBL SECTION4 RH".out.in_hp, out_in_wp => "DBVALVES"."TBL SECTION4 RH".out.in_wp, out_idle => "DBVALVES"."TBL SECTION4 RH".out.in_idle, out_status => "DBVALVES"."TBL SECTION4 RH".out.status)
   END_RUNG
   RUNG wire#powerrail
      Contact( "SIRIUS ESTOP" )
      Contact( "SIRIUS CURTAIN" )
   END_RUNG wire#w1
   // the same network as SCL:
   "INST TBL SECTION4 RH"(in_safety := "SIRIUS ESTOP" AND "SIRIUS CURTAIN",   // "3STATE_PISTON"
                          in_move_hp := "DBVALVES"."TBL SECTION4 RH".in.move_hp,
                          in_move_wp := "DBVALVES"."TBL SECTION4 RH".in.move_wp,
                          in_move_idle := "DBVALVES"."TBL SECTION4 RH".in.move_idle,
                          in_sensor_hp := "VSEN TBL SECTION4 RH HP UP",
                          in_sensor_wp := "VSEN TBL SECTION4 RH WP DOWN",
                          in_ez_hp := "VALVE TBL SECTION4 RH HP UP",
                          in_ez_wp := "VALVE TBL SECTION4 RH WP DOWN",
                          in_ez_idle := "DBVALVES"."TBL SECTION4 RH".test.IDLE_DUMMY,
                          out_in_hp => "DBVALVES"."TBL SECTION4 RH".out.in_hp,
                          out_in_wp => "DBVALVES"."TBL SECTION4 RH".out.in_wp,
                          out_idle => "DBVALVES"."TBL SECTION4 RH".out.in_idle,
                          out_status => "DBVALVES"."TBL SECTION4 RH".out.status);
END_REGION

REGION Network 140: [7] TBL SECTION5 LH
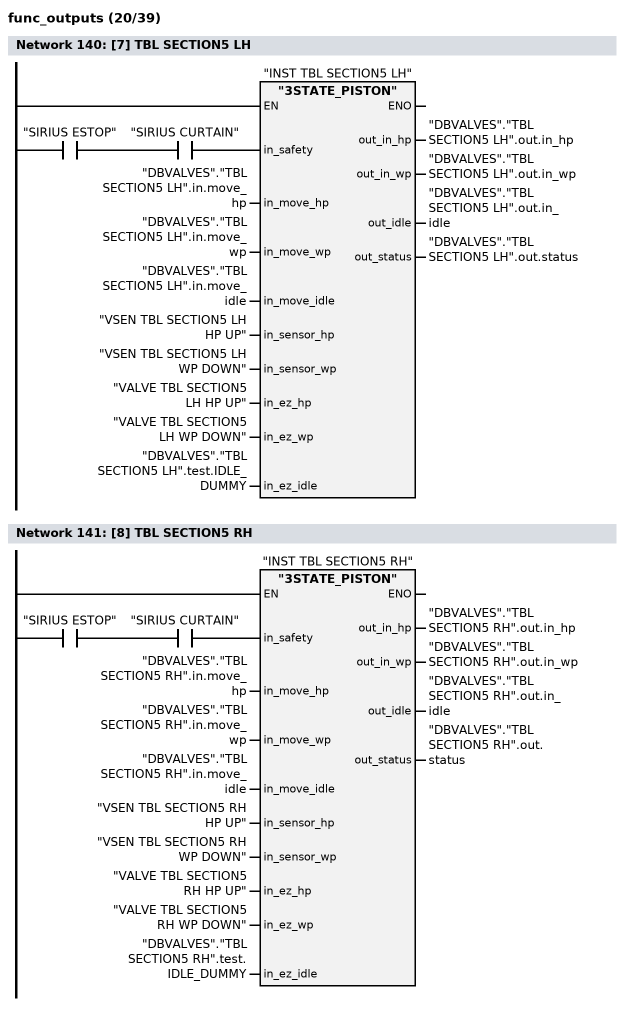
   RUNG wire#powerrail
      "INST TBL SECTION5 LH"(in_safety := wire#w1, in_move_hp := "DBVALVES"."TBL SECTION5 LH".in.move_hp, in_move_wp := "DBVALVES"."TBL SECTION5 LH".in.move_wp, in_move_idle := "DBVALVES"."TBL SECTION5 LH".in.move_idle, in_sensor_hp := "VSEN TBL SECTION5 LH HP UP", in_sensor_wp := "VSEN TBL SECTION5 LH WP DOWN", in_ez_hp := "VALVE TBL SECTION5 LH HP UP", in_ez_wp := "VALVE TBL SECTION5 LH WP DOWN", in_ez_idle := "DBVALVES"."TBL SECTION5 LH".test.IDLE_DUMMY, out_in_hp => "DBVALVES"."TBL SECTION5 LH".out.in_hp, out_in_wp => "DBVALVES"."TBL SECTION5 LH".out.in_wp, out_idle => "DBVALVES"."TBL SECTION5 LH".out.in_idle, out_status => "DBVALVES"."TBL SECTION5 LH".out.status)
   END_RUNG
   RUNG wire#powerrail
      Contact( "SIRIUS ESTOP" )
      Contact( "SIRIUS CURTAIN" )
   END_RUNG wire#w1
   // the same network as SCL:
   "INST TBL SECTION5 LH"(in_safety := "SIRIUS ESTOP" AND "SIRIUS CURTAIN",   // "3STATE_PISTON"
                          in_move_hp := "DBVALVES"."TBL SECTION5 LH".in.move_hp,
                          in_move_wp := "DBVALVES"."TBL SECTION5 LH".in.move_wp,
                          in_move_idle := "DBVALVES"."TBL SECTION5 LH".in.move_idle,
                          in_sensor_hp := "VSEN TBL SECTION5 LH HP UP",
                          in_sensor_wp := "VSEN TBL SECTION5 LH WP DOWN",
                          in_ez_hp := "VALVE TBL SECTION5 LH HP UP",
                          in_ez_wp := "VALVE TBL SECTION5 LH WP DOWN",
                          in_ez_idle := "DBVALVES"."TBL SECTION5 LH".test.IDLE_DUMMY,
                          out_in_hp => "DBVALVES"."TBL SECTION5 LH".out.in_hp,
                          out_in_wp => "DBVALVES"."TBL SECTION5 LH".out.in_wp,
                          out_idle => "DBVALVES"."TBL SECTION5 LH".out.in_idle,
                          out_status => "DBVALVES"."TBL SECTION5 LH".out.status);
END_REGION

REGION Network 141: [8] TBL SECTION5 RH
   RUNG wire#powerrail
      "INST TBL SECTION5 RH"(in_safety := wire#w1, in_move_hp := "DBVALVES"."TBL SECTION5 RH".in.move_hp, in_move_wp := "DBVALVES"."TBL SECTION5 RH".in.move_wp, in_move_idle := "DBVALVES"."TBL SECTION5 RH".in.move_idle, in_sensor_hp := "VSEN TBL SECTION5 RH HP UP", in_sensor_wp := "VSEN TBL SECTION5 RH WP DOWN", in_ez_hp := "VALVE TBL SECTION5 RH HP UP", in_ez_wp := "VALVE TBL SECTION5 RH WP DOWN", in_ez_idle := "DBVALVES"."TBL SECTION5 RH".test.IDLE_DUMMY, out_in_hp => "DBVALVES"."TBL SECTION5 RH".out.in_hp, out_in_wp => "DBVALVES"."TBL SECTION5 RH".out.in_wp, out_idle => "DBVALVES"."TBL SECTION5 RH".out.in_idle, out_status => "DBVALVES"."TBL SECTION5 RH".out.status)
   END_RUNG
   RUNG wire#powerrail
      Contact( "SIRIUS ESTOP" )
      Contact( "SIRIUS CURTAIN" )
   END_RUNG wire#w1
   // the same network as SCL:
   "INST TBL SECTION5 RH"(in_safety := "SIRIUS ESTOP" AND "SIRIUS CURTAIN",   // "3STATE_PISTON"
                          in_move_hp := "DBVALVES"."TBL SECTION5 RH".in.move_hp,
                          in_move_wp := "DBVALVES"."TBL SECTION5 RH".in.move_wp,
                          in_move_idle := "DBVALVES"."TBL SECTION5 RH".in.move_idle,
                          in_sensor_hp := "VSEN TBL SECTION5 RH HP UP",
                          in_sensor_wp := "VSEN TBL SECTION5 RH WP DOWN",
                          in_ez_hp := "VALVE TBL SECTION5 RH HP UP",
                          in_ez_wp := "VALVE TBL SECTION5 RH WP DOWN",
                          in_ez_idle := "DBVALVES"."TBL SECTION5 RH".test.IDLE_DUMMY,
                          out_in_hp => "DBVALVES"."TBL SECTION5 RH".out.in_hp,
                          out_in_wp => "DBVALVES"."TBL SECTION5 RH".out.in_wp,
                          out_idle => "DBVALVES"."TBL SECTION5 RH".out.in_idle,
                          out_status => "DBVALVES"."TBL SECTION5 RH".out.status);
END_REGION

REGION Network 142: [9] TBL POSITIONING LH
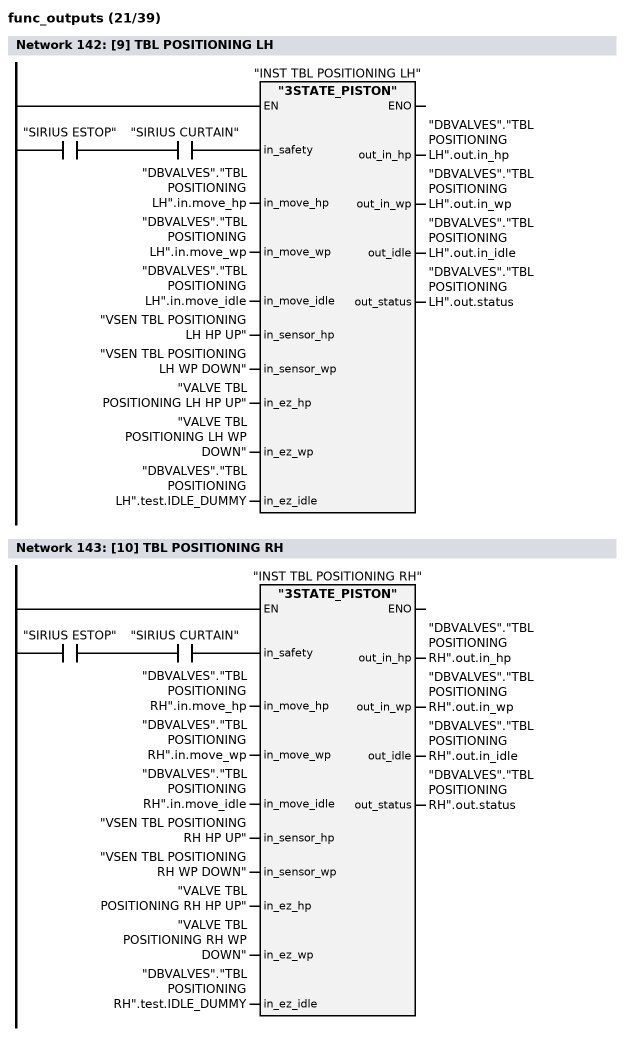
   RUNG wire#powerrail
      "INST TBL POSITIONING LH"(in_safety := wire#w1, in_move_hp := "DBVALVES"."TBL POSITIONING LH".in.move_hp, in_move_wp := "DBVALVES"."TBL POSITIONING LH".in.move_wp, in_move_idle := "DBVALVES"."TBL POSITIONING LH".in.move_idle, in_sensor_hp := "VSEN TBL POSITIONING LH HP UP", in_sensor_wp := "VSEN TBL POSITIONING LH WP DOWN", in_ez_hp := "VALVE TBL POSITIONING LH HP UP", in_ez_wp := "VALVE TBL POSITIONING LH WP DOWN", in_ez_idle := "DBVALVES"."TBL POSITIONING LH".test.IDLE_DUMMY, out_in_hp => "DBVALVES"."TBL POSITIONING LH".out.in_hp, out_in_wp => "DBVALVES"."TBL POSITIONING LH".out.in_wp, out_idle => "DBVALVES"."TBL POSITIONING LH".out.in_idle, out_status => "DBVALVES"."TBL POSITIONING LH".out.status)
   END_RUNG
   RUNG wire#powerrail
      Contact( "SIRIUS ESTOP" )
      Contact( "SIRIUS CURTAIN" )
   END_RUNG wire#w1
   // the same network as SCL:
   "INST TBL POSITIONING LH"(in_safety := "SIRIUS ESTOP" AND "SIRIUS CURTAIN",   // "3STATE_PISTON"
                           in_move_hp := "DBVALVES"."TBL POSITIONING LH".in.move_hp,
                           in_move_wp := "DBVALVES"."TBL POSITIONING LH".in.move_wp,
                           in_move_idle := "DBVALVES"."TBL POSITIONING LH".in.move_idle,
                           in_sensor_hp := "VSEN TBL POSITIONING LH HP UP",
                           in_sensor_wp := "VSEN TBL POSITIONING LH WP DOWN",
                           in_ez_hp := "VALVE TBL POSITIONING LH HP UP",
                           in_ez_wp := "VALVE TBL POSITIONING LH WP DOWN",
                           in_ez_idle := "DBVALVES"."TBL POSITIONING LH".test.IDLE_DUMMY,
                           out_in_hp => "DBVALVES"."TBL POSITIONING LH".out.in_hp,
                           out_in_wp => "DBVALVES"."TBL POSITIONING LH".out.in_wp,
                           out_idle => "DBVALVES"."TBL POSITIONING LH".out.in_idle,
                           out_status => "DBVALVES"."TBL POSITIONING LH".out.status);
END_REGION

REGION Network 143: [10] TBL POSITIONING RH
   RUNG wire#powerrail
      "INST TBL POSITIONING RH"(in_safety := wire#w1, in_move_hp := "DBVALVES"."TBL POSITIONING RH".in.move_hp, in_move_wp := "DBVALVES"."TBL POSITIONING RH".in.move_wp, in_move_idle := "DBVALVES"."TBL POSITIONING RH".in.move_idle, in_sensor_hp := "VSEN TBL POSITIONING RH HP UP", in_sensor_wp := "VSEN TBL POSITIONING RH WP DOWN", in_ez_hp := "VALVE TBL POSITIONING RH HP UP", in_ez_wp := "VALVE TBL POSITIONING RH WP DOWN", in_ez_idle := "DBVALVES"."TBL POSITIONING RH".test.IDLE_DUMMY, out_in_hp => "DBVALVES"."TBL POSITIONING RH".out.in_hp, out_in_wp => "DBVALVES"."TBL POSITIONING RH".out.in_wp, out_idle => "DBVALVES"."TBL POSITIONING RH".out.in_idle, out_status => "DBVALVES"."TBL POSITIONING RH".out.status)
   END_RUNG
   RUNG wire#powerrail
      Contact( "SIRIUS ESTOP" )
      Contact( "SIRIUS CURTAIN" )
   END_RUNG wire#w1
   // the same network as SCL:
   "INST TBL POSITIONING RH"(in_safety := "SIRIUS ESTOP" AND "SIRIUS CURTAIN",   // "3STATE_PISTON"
                           in_move_hp := "DBVALVES"."TBL POSITIONING RH".in.move_hp,
                           in_move_wp := "DBVALVES"."TBL POSITIONING RH".in.move_wp,
                           in_move_idle := "DBVALVES"."TBL POSITIONING RH".in.move_idle,
                           in_sensor_hp := "VSEN TBL POSITIONING RH HP UP",
                           in_sensor_wp := "VSEN TBL POSITIONING RH WP DOWN",
                           in_ez_hp := "VALVE TBL POSITIONING RH HP UP",
                           in_ez_wp := "VALVE TBL POSITIONING RH WP DOWN",
                           in_ez_idle := "DBVALVES"."TBL POSITIONING RH".test.IDLE_DUMMY,
                           out_in_hp => "DBVALVES"."TBL POSITIONING RH".out.in_hp,
                           out_in_wp => "DBVALVES"."TBL POSITIONING RH".out.in_wp,
                           out_idle => "DBVALVES"."TBL POSITIONING RH".out.in_idle,
                           out_status => "DBVALVES"."TBL POSITIONING RH".out.status);
END_REGION

REGION Network 144: [11] TBL PIN LH
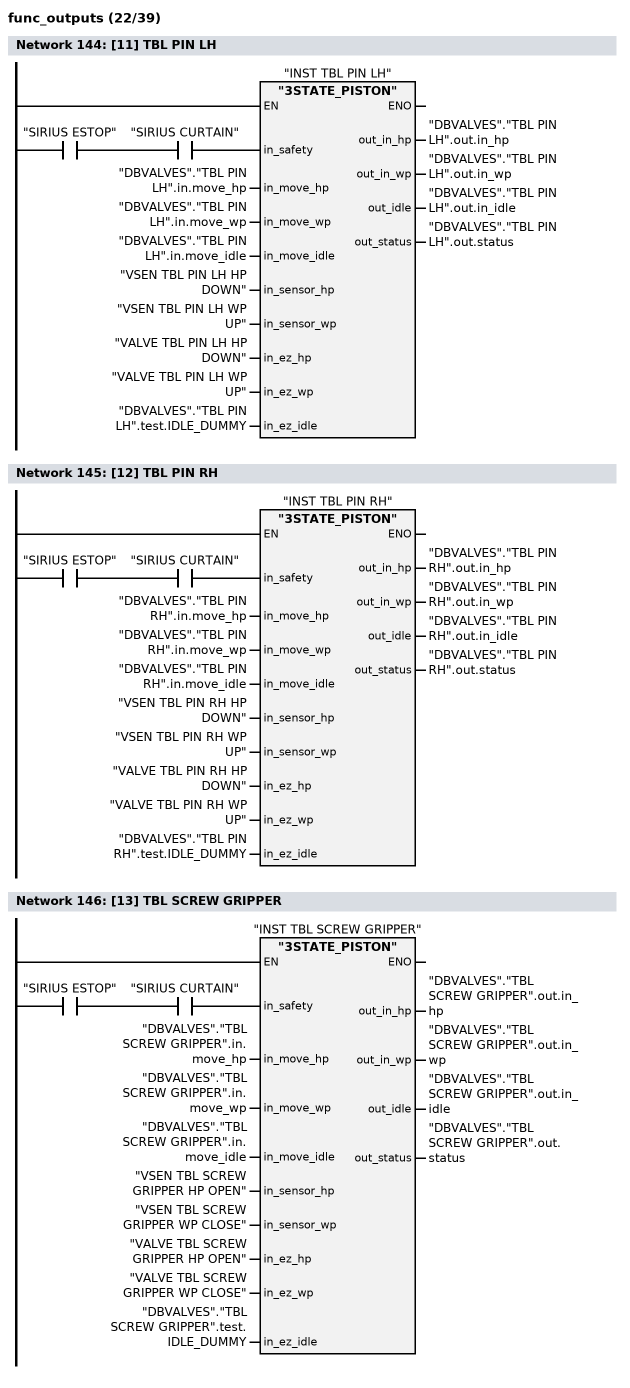
   RUNG wire#powerrail
      "INST TBL PIN LH"(in_safety := wire#w1, in_move_hp := "DBVALVES"."TBL PIN LH".in.move_hp, in_move_wp := "DBVALVES"."TBL PIN LH".in.move_wp, in_move_idle := "DBVALVES"."TBL PIN LH".in.move_idle, in_sensor_hp := "VSEN TBL PIN LH HP DOWN", in_sensor_wp := "VSEN TBL PIN LH WP UP", in_ez_hp := "VALVE TBL PIN LH HP DOWN", in_ez_wp := "VALVE TBL PIN LH WP UP", in_ez_idle := "DBVALVES"."TBL PIN LH".test.IDLE_DUMMY, out_in_hp => "DBVALVES"."TBL PIN LH".out.in_hp, out_in_wp => "DBVALVES"."TBL PIN LH".out.in_wp, out_idle => "DBVALVES"."TBL PIN LH".out.in_idle, out_status => "DBVALVES"."TBL PIN LH".out.status)
   END_RUNG
   RUNG wire#powerrail
      Contact( "SIRIUS ESTOP" )
      Contact( "SIRIUS CURTAIN" )
   END_RUNG wire#w1
   // the same network as SCL:
   "INST TBL PIN LH"(in_safety := "SIRIUS ESTOP" AND "SIRIUS CURTAIN",   // "3STATE_PISTON"
                     in_move_hp := "DBVALVES"."TBL PIN LH".in.move_hp,
                     in_move_wp := "DBVALVES"."TBL PIN LH".in.move_wp,
                     in_move_idle := "DBVALVES"."TBL PIN LH".in.move_idle,
                     in_sensor_hp := "VSEN TBL PIN LH HP DOWN",
                     in_sensor_wp := "VSEN TBL PIN LH WP UP",
                     in_ez_hp := "VALVE TBL PIN LH HP DOWN",
                     in_ez_wp := "VALVE TBL PIN LH WP UP",
                     in_ez_idle := "DBVALVES"."TBL PIN LH".test.IDLE_DUMMY,
                     out_in_hp => "DBVALVES"."TBL PIN LH".out.in_hp,
                     out_in_wp => "DBVALVES"."TBL PIN LH".out.in_wp,
                     out_idle => "DBVALVES"."TBL PIN LH".out.in_idle,
                     out_status => "DBVALVES"."TBL PIN LH".out.status);
END_REGION

REGION Network 145: [12] TBL PIN RH
   RUNG wire#powerrail
      "INST TBL PIN RH"(in_safety := wire#w1, in_move_hp := "DBVALVES"."TBL PIN RH".in.move_hp, in_move_wp := "DBVALVES"."TBL PIN RH".in.move_wp, in_move_idle := "DBVALVES"."TBL PIN RH".in.move_idle, in_sensor_hp := "VSEN TBL PIN RH HP DOWN", in_sensor_wp := "VSEN TBL PIN RH WP UP", in_ez_hp := "VALVE TBL PIN RH HP DOWN", in_ez_wp := "VALVE TBL PIN RH WP UP", in_ez_idle := "DBVALVES"."TBL PIN RH".test.IDLE_DUMMY, out_in_hp => "DBVALVES"."TBL PIN RH".out.in_hp, out_in_wp => "DBVALVES"."TBL PIN RH".out.in_wp, out_idle => "DBVALVES"."TBL PIN RH".out.in_idle, out_status => "DBVALVES"."TBL PIN RH".out.status)
   END_RUNG
   RUNG wire#powerrail
      Contact( "SIRIUS ESTOP" )
      Contact( "SIRIUS CURTAIN" )
   END_RUNG wire#w1
   // the same network as SCL:
   "INST TBL PIN RH"(in_safety := "SIRIUS ESTOP" AND "SIRIUS CURTAIN",   // "3STATE_PISTON"
                     in_move_hp := "DBVALVES"."TBL PIN RH".in.move_hp,
                     in_move_wp := "DBVALVES"."TBL PIN RH".in.move_wp,
                     in_move_idle := "DBVALVES"."TBL PIN RH".in.move_idle,
                     in_sensor_hp := "VSEN TBL PIN RH HP DOWN",
                     in_sensor_wp := "VSEN TBL PIN RH WP UP",
                     in_ez_hp := "VALVE TBL PIN RH HP DOWN",
                     in_ez_wp := "VALVE TBL PIN RH WP UP",
                     in_ez_idle := "DBVALVES"."TBL PIN RH".test.IDLE_DUMMY,
                     out_in_hp => "DBVALVES"."TBL PIN RH".out.in_hp,
                     out_in_wp => "DBVALVES"."TBL PIN RH".out.in_wp,
                     out_idle => "DBVALVES"."TBL PIN RH".out.in_idle,
                     out_status => "DBVALVES"."TBL PIN RH".out.status);
END_REGION

REGION Network 146: [13] TBL SCREW GRIPPER
   RUNG wire#powerrail
      "INST TBL SCREW GRIPPER"(in_safety := wire#w1, in_move_hp := "DBVALVES"."TBL SCREW GRIPPER".in.move_hp, in_move_wp := "DBVALVES"."TBL SCREW GRIPPER".in.move_wp, in_move_idle := "DBVALVES"."TBL SCREW GRIPPER".in.move_idle, in_sensor_hp := "VSEN TBL SCREW GRIPPER HP OPEN", in_sensor_wp := "VSEN TBL SCREW GRIPPER WP CLOSE", in_ez_hp := "VALVE TBL SCREW GRIPPER HP OPEN", in_ez_wp := "VALVE TBL SCREW GRIPPER WP CLOSE", in_ez_idle := "DBVALVES"."TBL SCREW GRIPPER".test.IDLE_DUMMY, out_in_hp => "DBVALVES"."TBL SCREW GRIPPER".out.in_hp, out_in_wp => "DBVALVES"."TBL SCREW GRIPPER".out.in_wp, out_idle => "DBVALVES"."TBL SCREW GRIPPER".out.in_idle, out_status => "DBVALVES"."TBL SCREW GRIPPER".out.status)
   END_RUNG
   RUNG wire#powerrail
      Contact( "SIRIUS ESTOP" )
      Contact( "SIRIUS CURTAIN" )
   END_RUNG wire#w1
   // the same network as SCL:
   "INST TBL SCREW GRIPPER"(in_safety := "SIRIUS ESTOP" AND "SIRIUS CURTAIN",   // "3STATE_PISTON"
                           in_move_hp := "DBVALVES"."TBL SCREW GRIPPER".in.move_hp,
                           in_move_wp := "DBVALVES"."TBL SCREW GRIPPER".in.move_wp,
                           in_move_idle := "DBVALVES"."TBL SCREW GRIPPER".in.move_idle,
                           in_sensor_hp := "VSEN TBL SCREW GRIPPER HP OPEN",
                           in_sensor_wp := "VSEN TBL SCREW GRIPPER WP CLOSE",
                           in_ez_hp := "VALVE TBL SCREW GRIPPER HP OPEN",
                           in_ez_wp := "VALVE TBL SCREW GRIPPER WP CLOSE",
                           in_ez_idle := "DBVALVES"."TBL SCREW GRIPPER".test.IDLE_DUMMY,
                           out_in_hp => "DBVALVES"."TBL SCREW GRIPPER".out.in_hp,
                           out_in_wp => "DBVALVES"."TBL SCREW GRIPPER".out.in_wp,
                           out_idle => "DBVALVES"."TBL SCREW GRIPPER".out.in_idle,
                           out_status => "DBVALVES"."TBL SCREW GRIPPER".out.status);
END_REGION

REGION Network 147: [14] TBL WRAP GRIPPER
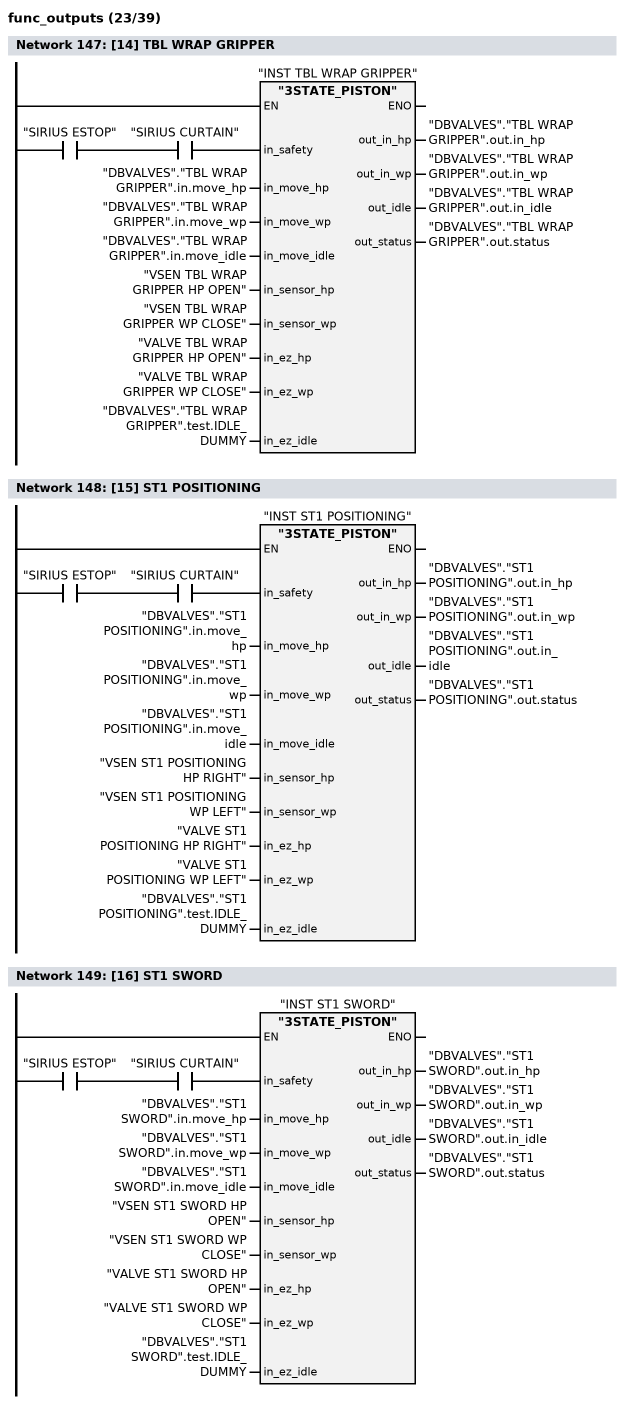
   RUNG wire#powerrail
      "INST TBL WRAP GRIPPER"(in_safety := wire#w1, in_move_hp := "DBVALVES"."TBL WRAP GRIPPER".in.move_hp, in_move_wp := "DBVALVES"."TBL WRAP GRIPPER".in.move_wp, in_move_idle := "DBVALVES"."TBL WRAP GRIPPER".in.move_idle, in_sensor_hp := "VSEN TBL WRAP GRIPPER HP OPEN", in_sensor_wp := "VSEN TBL WRAP GRIPPER WP CLOSE", in_ez_hp := "VALVE TBL WRAP GRIPPER HP OPEN", in_ez_wp := "VALVE TBL WRAP GRIPPER WP CLOSE", in_ez_idle := "DBVALVES"."TBL WRAP GRIPPER".test.IDLE_DUMMY, out_in_hp => "DBVALVES"."TBL WRAP GRIPPER".out.in_hp, out_in_wp => "DBVALVES"."TBL WRAP GRIPPER".out.in_wp, out_idle => "DBVALVES"."TBL WRAP GRIPPER".out.in_idle, out_status => "DBVALVES"."TBL WRAP GRIPPER".out.status)
   END_RUNG
   RUNG wire#powerrail
      Contact( "SIRIUS ESTOP" )
      Contact( "SIRIUS CURTAIN" )
   END_RUNG wire#w1
   // the same network as SCL:
   "INST TBL WRAP GRIPPER"(in_safety := "SIRIUS ESTOP" AND "SIRIUS CURTAIN",   // "3STATE_PISTON"
                           in_move_hp := "DBVALVES"."TBL WRAP GRIPPER".in.move_hp,
                           in_move_wp := "DBVALVES"."TBL WRAP GRIPPER".in.move_wp,
                           in_move_idle := "DBVALVES"."TBL WRAP GRIPPER".in.move_idle,
                           in_sensor_hp := "VSEN TBL WRAP GRIPPER HP OPEN",
                           in_sensor_wp := "VSEN TBL WRAP GRIPPER WP CLOSE",
                           in_ez_hp := "VALVE TBL WRAP GRIPPER HP OPEN",
                           in_ez_wp := "VALVE TBL WRAP GRIPPER WP CLOSE",
                           in_ez_idle := "DBVALVES"."TBL WRAP GRIPPER".test.IDLE_DUMMY,
                           out_in_hp => "DBVALVES"."TBL WRAP GRIPPER".out.in_hp,
                           out_in_wp => "DBVALVES"."TBL WRAP GRIPPER".out.in_wp,
                           out_idle => "DBVALVES"."TBL WRAP GRIPPER".out.in_idle,
                           out_status => "DBVALVES"."TBL WRAP GRIPPER".out.status);
END_REGION

REGION Network 148: [15] ST1 POSITIONING
   RUNG wire#powerrail
      "INST ST1 POSITIONING"(in_safety := wire#w1, in_move_hp := "DBVALVES"."ST1 POSITIONING".in.move_hp, in_move_wp := "DBVALVES"."ST1 POSITIONING".in.move_wp, in_move_idle := "DBVALVES"."ST1 POSITIONING".in.move_idle, in_sensor_hp := "VSEN ST1 POSITIONING HP RIGHT", in_sensor_wp := "VSEN ST1 POSITIONING WP LEFT", in_ez_hp := "VALVE ST1 POSITIONING HP RIGHT", in_ez_wp := "VALVE ST1 POSITIONING WP LEFT", in_ez_idle := "DBVALVES"."ST1 POSITIONING".test.IDLE_DUMMY, out_in_hp => "DBVALVES"."ST1 POSITIONING".out.in_hp, out_in_wp => "DBVALVES"."ST1 POSITIONING".out.in_wp, out_idle => "DBVALVES"."ST1 POSITIONING".out.in_idle, out_status => "DBVALVES"."ST1 POSITIONING".out.status)
   END_RUNG
   RUNG wire#powerrail
      Contact( "SIRIUS ESTOP" )
      Contact( "SIRIUS CURTAIN" )
   END_RUNG wire#w1
   // the same network as SCL:
   "INST ST1 POSITIONING"(in_safety := "SIRIUS ESTOP" AND "SIRIUS CURTAIN",   // "3STATE_PISTON"
                          in_move_hp := "DBVALVES"."ST1 POSITIONING".in.move_hp,
                          in_move_wp := "DBVALVES"."ST1 POSITIONING".in.move_wp,
                          in_move_idle := "DBVALVES"."ST1 POSITIONING".in.move_idle,
                          in_sensor_hp := "VSEN ST1 POSITIONING HP RIGHT",
                          in_sensor_wp := "VSEN ST1 POSITIONING WP LEFT",
                          in_ez_hp := "VALVE ST1 POSITIONING HP RIGHT",
                          in_ez_wp := "VALVE ST1 POSITIONING WP LEFT",
                          in_ez_idle := "DBVALVES"."ST1 POSITIONING".test.IDLE_DUMMY,
                          out_in_hp => "DBVALVES"."ST1 POSITIONING".out.in_hp,
                          out_in_wp => "DBVALVES"."ST1 POSITIONING".out.in_wp,
                          out_idle => "DBVALVES"."ST1 POSITIONING".out.in_idle,
                          out_status => "DBVALVES"."ST1 POSITIONING".out.status);
END_REGION

REGION Network 149: [16] ST1 SWORD
   RUNG wire#powerrail
      "INST ST1 SWORD"(in_safety := wire#w1, in_move_hp := "DBVALVES"."ST1 SWORD".in.move_hp, in_move_wp := "DBVALVES"."ST1 SWORD".in.move_wp, in_move_idle := "DBVALVES"."ST1 SWORD".in.move_idle, in_sensor_hp := "VSEN ST1 SWORD HP OPEN", in_sensor_wp := "VSEN ST1 SWORD WP CLOSE", in_ez_hp := "VALVE ST1 SWORD HP OPEN", in_ez_wp := "VALVE ST1 SWORD WP CLOSE", in_ez_idle := "DBVALVES"."ST1 SWORD".test.IDLE_DUMMY, out_in_hp => "DBVALVES"."ST1 SWORD".out.in_hp, out_in_wp => "DBVALVES"."ST1 SWORD".out.in_wp, out_idle => "DBVALVES"."ST1 SWORD".out.in_idle, out_status => "DBVALVES"."ST1 SWORD".out.status)
   END_RUNG
   RUNG wire#powerrail
      Contact( "SIRIUS ESTOP" )
      Contact( "SIRIUS CURTAIN" )
   END_RUNG wire#w1
   // the same network as SCL:
   "INST ST1 SWORD"(in_safety := "SIRIUS ESTOP" AND "SIRIUS CURTAIN",   // "3STATE_PISTON"
                    in_move_hp := "DBVALVES"."ST1 SWORD".in.move_hp,
                    in_move_wp := "DBVALVES"."ST1 SWORD".in.move_wp,
                    in_move_idle := "DBVALVES"."ST1 SWORD".in.move_idle,
                    in_sensor_hp := "VSEN ST1 SWORD HP OPEN",
                    in_sensor_wp := "VSEN ST1 SWORD WP CLOSE",
                    in_ez_hp := "VALVE ST1 SWORD HP OPEN",
                    in_ez_wp := "VALVE ST1 SWORD WP CLOSE",
                    in_ez_idle := "DBVALVES"."ST1 SWORD".test.IDLE_DUMMY,
                    out_in_hp => "DBVALVES"."ST1 SWORD".out.in_hp,
                    out_in_wp => "DBVALVES"."ST1 SWORD".out.in_wp,
                    out_idle => "DBVALVES"."ST1 SWORD".out.in_idle,
                    out_status => "DBVALVES"."ST1 SWORD".out.status);
END_REGION

REGION Network 150: [17] ST2 POSITIONING
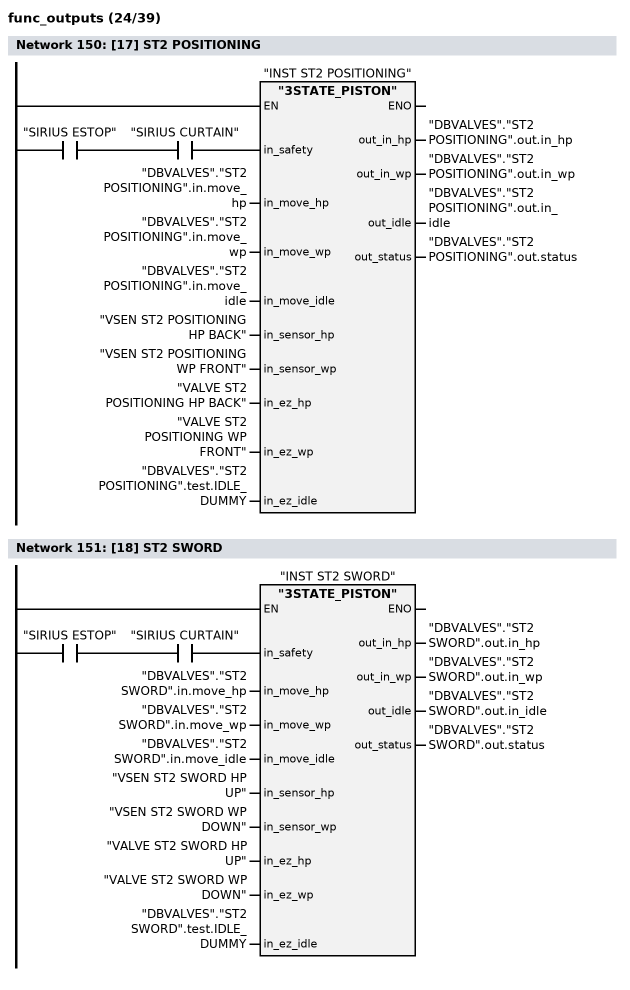
   RUNG wire#powerrail
      "INST ST2 POSITIONING"(in_safety := wire#w1, in_move_hp := "DBVALVES"."ST2 POSITIONING".in.move_hp, in_move_wp := "DBVALVES"."ST2 POSITIONING".in.move_wp, in_move_idle := "DBVALVES"."ST2 POSITIONING".in.move_idle, in_sensor_hp := "VSEN ST2 POSITIONING HP BACK", in_sensor_wp := "VSEN ST2 POSITIONING WP FRONT", in_ez_hp := "VALVE ST2 POSITIONING HP BACK", in_ez_wp := "VALVE ST2 POSITIONING WP FRONT", in_ez_idle := "DBVALVES"."ST2 POSITIONING".test.IDLE_DUMMY, out_in_hp => "DBVALVES"."ST2 POSITIONING".out.in_hp, out_in_wp => "DBVALVES"."ST2 POSITIONING".out.in_wp, out_idle => "DBVALVES"."ST2 POSITIONING".out.in_idle, out_status => "DBVALVES"."ST2 POSITIONING".out.status)
   END_RUNG
   RUNG wire#powerrail
      Contact( "SIRIUS ESTOP" )
      Contact( "SIRIUS CURTAIN" )
   END_RUNG wire#w1
   // the same network as SCL:
   "INST ST2 POSITIONING"(in_safety := "SIRIUS ESTOP" AND "SIRIUS CURTAIN",   // "3STATE_PISTON"
                          in_move_hp := "DBVALVES"."ST2 POSITIONING".in.move_hp,
                          in_move_wp := "DBVALVES"."ST2 POSITIONING".in.move_wp,
                          in_move_idle := "DBVALVES"."ST2 POSITIONING".in.move_idle,
                          in_sensor_hp := "VSEN ST2 POSITIONING HP BACK",
                          in_sensor_wp := "VSEN ST2 POSITIONING WP FRONT",
                          in_ez_hp := "VALVE ST2 POSITIONING HP BACK",
                          in_ez_wp := "VALVE ST2 POSITIONING WP FRONT",
                          in_ez_idle := "DBVALVES"."ST2 POSITIONING".test.IDLE_DUMMY,
                          out_in_hp => "DBVALVES"."ST2 POSITIONING".out.in_hp,
                          out_in_wp => "DBVALVES"."ST2 POSITIONING".out.in_wp,
                          out_idle => "DBVALVES"."ST2 POSITIONING".out.in_idle,
                          out_status => "DBVALVES"."ST2 POSITIONING".out.status);
END_REGION

REGION Network 151: [18] ST2 SWORD
   RUNG wire#powerrail
      "INST ST2 SWORD"(in_safety := wire#w1, in_move_hp := "DBVALVES"."ST2 SWORD".in.move_hp, in_move_wp := "DBVALVES"."ST2 SWORD".in.move_wp, in_move_idle := "DBVALVES"."ST2 SWORD".in.move_idle, in_sensor_hp := "VSEN ST2 SWORD HP UP", in_sensor_wp := "VSEN ST2 SWORD WP DOWN", in_ez_hp := "VALVE ST2 SWORD HP UP", in_ez_wp := "VALVE ST2 SWORD WP DOWN", in_ez_idle := "DBVALVES"."ST2 SWORD".test.IDLE_DUMMY, out_in_hp => "DBVALVES"."ST2 SWORD".out.in_hp, out_in_wp => "DBVALVES"."ST2 SWORD".out.in_wp, out_idle => "DBVALVES"."ST2 SWORD".out.in_idle, out_status => "DBVALVES"."ST2 SWORD".out.status)
   END_RUNG
   RUNG wire#powerrail
      Contact( "SIRIUS ESTOP" )
      Contact( "SIRIUS CURTAIN" )
   END_RUNG wire#w1
   // the same network as SCL:
   "INST ST2 SWORD"(in_safety := "SIRIUS ESTOP" AND "SIRIUS CURTAIN",   // "3STATE_PISTON"
                    in_move_hp := "DBVALVES"."ST2 SWORD".in.move_hp,
                    in_move_wp := "DBVALVES"."ST2 SWORD".in.move_wp,
                    in_move_idle := "DBVALVES"."ST2 SWORD".in.move_idle,
                    in_sensor_hp := "VSEN ST2 SWORD HP UP",
                    in_sensor_wp := "VSEN ST2 SWORD WP DOWN",
                    in_ez_hp := "VALVE ST2 SWORD HP UP",
                    in_ez_wp := "VALVE ST2 SWORD WP DOWN",
                    in_ez_idle := "DBVALVES"."ST2 SWORD".test.IDLE_DUMMY,
                    out_in_hp => "DBVALVES"."ST2 SWORD".out.in_hp,
                    out_in_wp => "DBVALVES"."ST2 SWORD".out.in_wp,
                    out_idle => "DBVALVES"."ST2 SWORD".out.in_idle,
                    out_status => "DBVALVES"."ST2 SWORD".out.status);
END_REGION

REGION Network 152: [19] ST3 POSITIONING
